// LMC_PacDrive/Application/TemplateFullProgrammingFramework/Visualization/Multicarrier/Vis_Positions_31_60
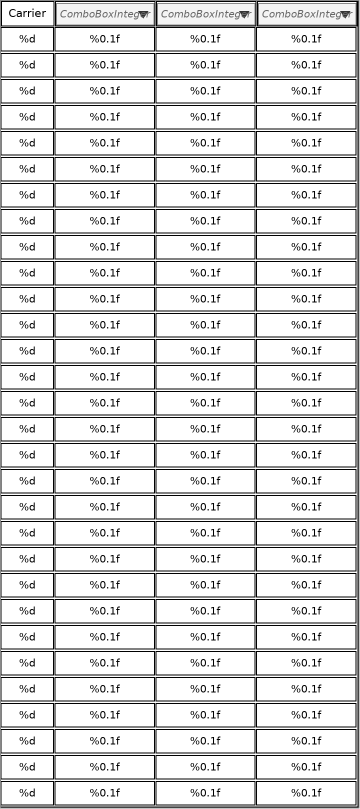
VISUALIZATION Vis_Positions_31_60  // 360x809
    Rectangle (0,0 358x807)
    Rectangle (55,1 100x25), "Position", invisible if: not SR_MultiCarriermodule.xInitSuccessful
    Rectangle (156,1 100x25), "Gap In Front", invisible if: not SR_MultiCarriermodule.xInitSuccessful
    Rectangle (257,1 100x25), "Gap Behind", invisible if: not SR_MultiCarriermodule.xInitSuccessful
    Rectangle (1,1 53x25), "Carrier", invisible if: not SR_MultiCarriermodule.xInitSuccessful
    Frame (0,27 358x26), invisible if: SR_MulticarrierModule.ifMulticarrier.ifFeedback.ifFeedbackConfiguration.udiNumberOfCarriers < 31 OR NOT SR_MultiCarriermodule.xInitSuccessful
        shows FR_CarDist(i_ifCarrierFeedback := SR_MultiCarrierModule.aifVisFeedback[31])
    Frame (0,53 358x26), invisible if: SR_MulticarrierModule.ifMulticarrier.ifFeedback.ifFeedbackConfiguration.udiNumberOfCarriers < 32 OR NOT SR_MultiCarriermodule.xInitSuccessful
        shows FR_CarDist(i_ifCarrierFeedback := SR_MultiCarrierModule.aifVisFeedback[32])
    Frame (0,79 358x26), invisible if: SR_MulticarrierModule.ifMulticarrier.ifFeedback.ifFeedbackConfiguration.udiNumberOfCarriers < 33 OR NOT SR_MultiCarriermodule.xInitSuccessful
        shows FR_CarDist(i_ifCarrierFeedback := SR_MultiCarrierModule.aifVisFeedback[33])
    Frame (0,105 358x26), invisible if: SR_MulticarrierModule.ifMulticarrier.ifFeedback.ifFeedbackConfiguration.udiNumberOfCarriers < 34 OR NOT SR_MultiCarriermodule.xInitSuccessful
        shows FR_CarDist(i_ifCarrierFeedback := SR_MultiCarrierModule.aifVisFeedback[34])
    Frame (0,131 358x26), invisible if: SR_MulticarrierModule.ifMulticarrier.ifFeedback.ifFeedbackConfiguration.udiNumberOfCarriers < 35 OR NOT SR_MultiCarriermodule.xInitSuccessful
        shows FR_CarDist(i_ifCarrierFeedback := SR_MultiCarrierModule.aifVisFeedback[35])
    Frame (0,157 358x26), invisible if: SR_MulticarrierModule.ifMulticarrier.ifFeedback.ifFeedbackConfiguration.udiNumberOfCarriers < 36 OR NOT SR_MultiCarriermodule.xInitSuccessful
        shows FR_CarDist(i_ifCarrierFeedback := SR_MultiCarrierModule.aifVisFeedback[36])
    Frame (0,183 358x26), invisible if: SR_MulticarrierModule.ifMulticarrier.ifFeedback.ifFeedbackConfiguration.udiNumberOfCarriers < 37 OR NOT SR_MultiCarriermodule.xInitSuccessful
        shows FR_CarDist(i_ifCarrierFeedback := SR_MultiCarrierModule.aifVisFeedback[37])
    Frame (0,209 358x26), invisible if: SR_MulticarrierModule.ifMulticarrier.ifFeedback.ifFeedbackConfiguration.udiNumberOfCarriers < 38 OR NOT SR_MultiCarriermodule.xInitSuccessful
        shows FR_CarDist(i_ifCarrierFeedback := SR_MultiCarrierModule.aifVisFeedback[38])
    Frame (0,235 358x26), invisible if: SR_MulticarrierModule.ifMulticarrier.ifFeedback.ifFeedbackConfiguration.udiNumberOfCarriers < 39 OR NOT SR_MultiCarriermodule.xInitSuccessful
        shows FR_CarDist(i_ifCarrierFeedback := SR_MultiCarrierModule.aifVisFeedback[39])
    Frame (0,261 358x26), invisible if: SR_MulticarrierModule.ifMulticarrier.ifFeedback.ifFeedbackConfiguration.udiNumberOfCarriers < 40 OR NOT SR_MultiCarriermodule.xInitSuccessful
        shows FR_CarDist(i_ifCarrierFeedback := SR_MultiCarrierModule.aifVisFeedback[40])
    ComboBoxInteger (258,3 98x22), tooltip "RefTrackPosition RefPosition Gap to Carrier in front Distance to Carrier in front Gap to Carrier behind Distance to Carrier behind", variable: SR_MulticarrierModule.etVisPosColumn3, text list: 'TextList_VisPositions'
    ComboBoxInteger (157,3 98x22), tooltip "RefTrackPosition RefPosition Gap to Carrier in front Distance to Carrier in front Gap to Carrier behind Distance to Carrier behind", variable: SR_MulticarrierModule.etVisPosColumn2, text list: 'TextList_VisPositions'
    ComboBoxInteger (56,3 98x22), tooltip "RefTrackPosition RefPosition Gap to Carrier in front Distance to Carrier in front Gap to Carrier behind Distance to Carrier behind", variable: SR_MulticarrierModule.etVisPosColumn1, text list: 'TextList_VisPositions'
    Frame (0,495 358x26), invisible if: SR_MulticarrierModule.ifMulticarrier.ifFeedback.ifFeedbackConfiguration.udiNumberOfCarriers < 50 OR NOT SR_MultiCarriermodule.xInitSuccessful
        shows FR_CarDist(i_ifCarrierFeedback := SR_MultiCarrierModule.aifVisFeedback[50])
    Frame (0,547 358x26), invisible if: SR_MulticarrierModule.ifMulticarrier.ifFeedback.ifFeedbackConfiguration.udiNumberOfCarriers < 51 OR NOT SR_MultiCarriermodule.xInitSuccessful
        shows FR_CarDist(i_ifCarrierFeedback := SR_MultiCarrierModule.aifVisFeedback[51])
    Frame (0,573 358x26), invisible if: SR_MulticarrierModule.ifMulticarrier.ifFeedback.ifFeedbackConfiguration.udiNumberOfCarriers < 52 OR NOT SR_MultiCarriermodule.xInitSuccessful
        shows FR_CarDist(i_ifCarrierFeedback := SR_MultiCarrierModule.aifVisFeedback[52])
    Frame (0,599 358x26), invisible if: SR_MulticarrierModule.ifMulticarrier.ifFeedback.ifFeedbackConfiguration.udiNumberOfCarriers < 53 OR NOT SR_MultiCarriermodule.xInitSuccessful
        shows FR_CarDist(i_ifCarrierFeedback := SR_MultiCarrierModule.aifVisFeedback[53])
    Frame (0,625 358x26), invisible if: SR_MulticarrierModule.ifMulticarrier.ifFeedback.ifFeedbackConfiguration.udiNumberOfCarriers < 54 OR NOT SR_MultiCarriermodule.xInitSuccessful
        shows FR_CarDist(i_ifCarrierFeedback := SR_MultiCarrierModule.aifVisFeedback[54])
    Frame (0,651 358x26), invisible if: SR_MulticarrierModule.ifMulticarrier.ifFeedback.ifFeedbackConfiguration.udiNumberOfCarriers < 55 OR NOT SR_MultiCarriermodule.xInitSuccessful
        shows FR_CarDist(i_ifCarrierFeedback := SR_MultiCarrierModule.aifVisFeedback[55])
    Frame (0,677 358x26), invisible if: SR_MulticarrierModule.ifMulticarrier.ifFeedback.ifFeedbackConfiguration.udiNumberOfCarriers < 56 OR NOT SR_MultiCarriermodule.xInitSuccessful
        shows FR_CarDist(i_ifCarrierFeedback := SR_MultiCarrierModule.aifVisFeedback[56])
    Frame (0,703 358x26), invisible if: SR_MulticarrierModule.ifMulticarrier.ifFeedback.ifFeedbackConfiguration.udiNumberOfCarriers < 57 OR NOT SR_MultiCarriermodule.xInitSuccessful
        shows FR_CarDist(i_ifCarrierFeedback := SR_MultiCarrierModule.aifVisFeedback[57])
    Frame (0,729 358x26), invisible if: SR_MulticarrierModule.ifMulticarrier.ifFeedback.ifFeedbackConfiguration.udiNumberOfCarriers < 58 OR NOT SR_MultiCarriermodule.xInitSuccessful
        shows FR_CarDist(i_ifCarrierFeedback := SR_MultiCarrierModule.aifVisFeedback[58])
    Frame (0,755 358x26), invisible if: SR_MulticarrierModule.ifMulticarrier.ifFeedback.ifFeedbackConfiguration.udiNumberOfCarriers < 59 OR NOT SR_MultiCarriermodule.xInitSuccessful
        shows FR_CarDist(i_ifCarrierFeedback := SR_MultiCarrierModule.aifVisFeedback[59])
    Frame (0,287 358x26), invisible if: SR_MulticarrierModule.ifMulticarrier.ifFeedback.ifFeedbackConfiguration.udiNumberOfCarriers < 41 OR NOT SR_MultiCarriermodule.xInitSuccessful
        shows FR_CarDist(i_ifCarrierFeedback := SR_MultiCarrierModule.aifVisFeedback[41])
    Frame (0,313 358x26), invisible if: SR_MulticarrierModule.ifMulticarrier.ifFeedback.ifFeedbackConfiguration.udiNumberOfCarriers < 42 OR NOT SR_MultiCarriermodule.xInitSuccessful
        shows FR_CarDist(i_ifCarrierFeedback := SR_MultiCarrierModule.aifVisFeedback[42])
    Frame (0,339 358x26), invisible if: SR_MulticarrierModule.ifMulticarrier.ifFeedback.ifFeedbackConfiguration.udiNumberOfCarriers < 43 OR NOT SR_MultiCarriermodule.xInitSuccessful
        shows FR_CarDist(i_ifCarrierFeedback := SR_MultiCarrierModule.aifVisFeedback[43])
    Frame (0,365 358x26), invisible if: SR_MulticarrierModule.ifMulticarrier.ifFeedback.ifFeedbackConfiguration.udiNumberOfCarriers < 44 OR NOT SR_MultiCarriermodule.xInitSuccessful
        shows FR_CarDist(i_ifCarrierFeedback := SR_MultiCarrierModule.aifVisFeedback[44])
    Frame (0,391 358x26), invisible if: SR_MulticarrierModule.ifMulticarrier.ifFeedback.ifFeedbackConfiguration.udiNumberOfCarriers < 45 OR NOT SR_MultiCarriermodule.xInitSuccessful
        shows FR_CarDist(i_ifCarrierFeedback := SR_MultiCarrierModule.aifVisFeedback[45])
    Frame (0,417 358x26), invisible if: SR_MulticarrierModule.ifMulticarrier.ifFeedback.ifFeedbackConfiguration.udiNumberOfCarriers < 46 OR NOT SR_MultiCarriermodule.xInitSuccessful
        shows FR_CarDist(i_ifCarrierFeedback := SR_MultiCarrierModule.aifVisFeedback[46])
    Frame (0,443 358x26), invisible if: SR_MulticarrierModule.ifMulticarrier.ifFeedback.ifFeedbackConfiguration.udiNumberOfCarriers < 47 OR NOT SR_MultiCarriermodule.xInitSuccessful
        shows FR_CarDist(i_ifCarrierFeedback := SR_MultiCarrierModule.aifVisFeedback[47])
    Frame (0,469 358x26), invisible if: SR_MulticarrierModule.ifMulticarrier.ifFeedback.ifFeedbackConfiguration.udiNumberOfCarriers < 48 OR NOT SR_MultiCarriermodule.xInitSuccessful
        shows FR_CarDist(i_ifCarrierFeedback := SR_MultiCarrierModule.aifVisFeedback[48])
    Frame (0,495 358x26), invisible if: SR_MulticarrierModule.ifMulticarrier.ifFeedback.ifFeedbackConfiguration.udiNumberOfCarriers < 49 OR NOT SR_MultiCarriermodule.xInitSuccessful
        shows FR_CarDist(i_ifCarrierFeedback := SR_MultiCarrierModule.aifVisFeedback[49])
    Frame (0,521 358x26), invisible if: SR_MulticarrierModule.ifMulticarrier.ifFeedback.ifFeedbackConfiguration.udiNumberOfCarriers < 50 OR NOT SR_MultiCarriermodule.xInitSuccessful
        shows FR_CarDist(i_ifCarrierFeedback := SR_MultiCarrierModule.aifVisFeedback[50])
    Frame (0,781 358x26), invisible if: SR_MulticarrierModule.ifMulticarrier.ifFeedback.ifFeedbackConfiguration.udiNumberOfCarriers < 60 OR NOT SR_MultiCarriermodule.xInitSuccessful
        shows FR_CarDist(i_ifCarrierFeedback := SR_MultiCarrierModule.aifVisFeedback[60])
END_VISUALIZATION

// LMC_PacDrive/Application/TemplateFullProgrammingFramework/Visualization/Multicarrier/Vis_Positions_61_90
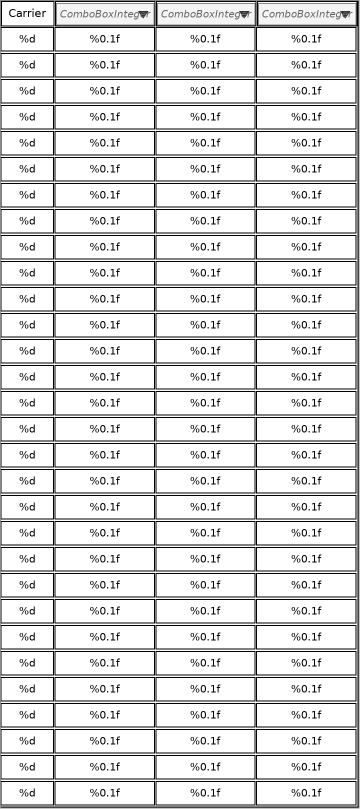
VISUALIZATION Vis_Positions_61_90  // 360x809
    Rectangle (0,0 358x807)
    Rectangle (55,1 100x25), "Position", invisible if: not SR_MultiCarriermodule.xInitSuccessful
    Rectangle (156,1 100x25), "Gap In Front", invisible if: not SR_MultiCarriermodule.xInitSuccessful
    Rectangle (257,1 100x25), "Gap Behind", invisible if: not SR_MultiCarriermodule.xInitSuccessful
    Rectangle (1,1 53x25), "Carrier", invisible if: not SR_MultiCarriermodule.xInitSuccessful
    Rectangle (55,1 100x25), "Position", invisible if: not SR_MultiCarriermodule.xInitSuccessful
    Rectangle (156,1 100x25), "Gap In Front", invisible if: not SR_MultiCarriermodule.xInitSuccessful
    Rectangle (257,1 100x25), "Gap Behind", invisible if: not SR_MultiCarriermodule.xInitSuccessful
    ComboBoxInteger (258,3 98x22), tooltip "RefTrackPosition RefPosition Gap to Carrier in front Distance to Carrier in front Gap to Carrier behind Distance to Carrier behind", variable: SR_MulticarrierModule.etVisPosColumn3, text list: 'TextList_VisPositions'
    ComboBoxInteger (157,3 98x22), tooltip "RefTrackPosition RefPosition Gap to Carrier in front Distance to Carrier in front Gap to Carrier behind Distance to Carrier behind", variable: SR_MulticarrierModule.etVisPosColumn2, text list: 'TextList_VisPositions'
    ComboBoxInteger (56,3 98x22), tooltip "RefTrackPosition RefPosition Gap to Carrier in front Distance to Carrier in front Gap to Carrier behind Distance to Carrier behind", variable: SR_MulticarrierModule.etVisPosColumn1, text list: 'TextList_VisPositions'
    Frame (0,27 358x26), invisible if: SR_MulticarrierModule.ifMulticarrier.ifFeedback.ifFeedbackConfiguration.udiNumberOfCarriers < 61 OR NOT SR_MultiCarriermodule.xInitSuccessful
        shows FR_CarDist(i_ifCarrierFeedback := SR_MultiCarrierModule.aifVisFeedback[61])
    Frame (0,261 358x26), invisible if: SR_MulticarrierModule.ifMulticarrier.ifFeedback.ifFeedbackConfiguration.udiNumberOfCarriers < 70 OR NOT SR_MultiCarriermodule.xInitSuccessful
        shows FR_CarDist(i_ifCarrierFeedback := SR_MultiCarrierModule.aifVisFeedback[70])
    Frame (0,53 358x26), invisible if: SR_MulticarrierModule.ifMulticarrier.ifFeedback.ifFeedbackConfiguration.udiNumberOfCarriers < 62 OR NOT SR_MultiCarriermodule.xInitSuccessful
        shows FR_CarDist(i_ifCarrierFeedback := SR_MultiCarrierModule.aifVisFeedback[62])
    Frame (0,105 358x26), invisible if: SR_MulticarrierModule.ifMulticarrier.ifFeedback.ifFeedbackConfiguration.udiNumberOfCarriers < 64 OR NOT SR_MultiCarriermodule.xInitSuccessful
        shows FR_CarDist(i_ifCarrierFeedback := SR_MultiCarrierModule.aifVisFeedback[64])
    Frame (0,131 358x26), invisible if: SR_MulticarrierModule.ifMulticarrier.ifFeedback.ifFeedbackConfiguration.udiNumberOfCarriers < 65 OR NOT SR_MultiCarriermodule.xInitSuccessful
        shows FR_CarDist(i_ifCarrierFeedback := SR_MultiCarrierModule.aifVisFeedback[65])
    Frame (0,157 358x26), invisible if: SR_MulticarrierModule.ifMulticarrier.ifFeedback.ifFeedbackConfiguration.udiNumberOfCarriers < 66 OR NOT SR_MultiCarriermodule.xInitSuccessful
        shows FR_CarDist(i_ifCarrierFeedback := SR_MultiCarrierModule.aifVisFeedback[66])
    Frame (0,209 358x26), invisible if: SR_MulticarrierModule.ifMulticarrier.ifFeedback.ifFeedbackConfiguration.udiNumberOfCarriers < 68 OR NOT SR_MultiCarriermodule.xInitSuccessful
        shows FR_CarDist(i_ifCarrierFeedback := SR_MultiCarrierModule.aifVisFeedback[68])
    Frame (0,235 358x26), invisible if: SR_MulticarrierModule.ifMulticarrier.ifFeedback.ifFeedbackConfiguration.udiNumberOfCarriers < 69 OR NOT SR_MultiCarriermodule.xInitSuccessful
        shows FR_CarDist(i_ifCarrierFeedback := SR_MultiCarrierModule.aifVisFeedback[69])
    Frame (0,287 358x26), invisible if: SR_MulticarrierModule.ifMulticarrier.ifFeedback.ifFeedbackConfiguration.udiNumberOfCarriers < 71 OR NOT SR_MultiCarriermodule.xInitSuccessful
        shows FR_CarDist(i_ifCarrierFeedback := SR_MultiCarrierModule.aifVisFeedback[71])
    Frame (0,313 358x26), invisible if: SR_MulticarrierModule.ifMulticarrier.ifFeedback.ifFeedbackConfiguration.udiNumberOfCarriers < 72 OR NOT SR_MultiCarriermodule.xInitSuccessful
        shows FR_CarDist(i_ifCarrierFeedback := SR_MultiCarrierModule.aifVisFeedback[72])
    Frame (0,339 358x26), invisible if: SR_MulticarrierModule.ifMulticarrier.ifFeedback.ifFeedbackConfiguration.udiNumberOfCarriers < 73 OR NOT SR_MultiCarriermodule.xInitSuccessful
        shows FR_CarDist(i_ifCarrierFeedback := SR_MultiCarrierModule.aifVisFeedback[73])
    Frame (0,365 358x26), invisible if: SR_MulticarrierModule.ifMulticarrier.ifFeedback.ifFeedbackConfiguration.udiNumberOfCarriers < 74 OR NOT SR_MultiCarriermodule.xInitSuccessful
        shows FR_CarDist(i_ifCarrierFeedback := SR_MultiCarrierModule.aifVisFeedback[74])
    Frame (0,391 358x26), invisible if: SR_MulticarrierModule.ifMulticarrier.ifFeedback.ifFeedbackConfiguration.udiNumberOfCarriers < 75 OR NOT SR_MultiCarriermodule.xInitSuccessful
        shows FR_CarDist(i_ifCarrierFeedback := SR_MultiCarrierModule.aifVisFeedback[75])
    Frame (0,417 358x26), invisible if: SR_MulticarrierModule.ifMulticarrier.ifFeedback.ifFeedbackConfiguration.udiNumberOfCarriers < 76 OR NOT SR_MultiCarriermodule.xInitSuccessful
        shows FR_CarDist(i_ifCarrierFeedback := SR_MultiCarrierModule.aifVisFeedback[76])
    Frame (0,443 358x26), invisible if: SR_MulticarrierModule.ifMulticarrier.ifFeedback.ifFeedbackConfiguration.udiNumberOfCarriers < 77 OR NOT SR_MultiCarriermodule.xInitSuccessful
        shows FR_CarDist(i_ifCarrierFeedback := SR_MultiCarrierModule.aifVisFeedback[77])
    Frame (0,469 358x26), invisible if: SR_MulticarrierModule.ifMulticarrier.ifFeedback.ifFeedbackConfiguration.udiNumberOfCarriers < 78 OR NOT SR_MultiCarriermodule.xInitSuccessful
        shows FR_CarDist(i_ifCarrierFeedback := SR_MultiCarrierModule.aifVisFeedback[78])
    Frame (0,495 358x26), invisible if: SR_MulticarrierModule.ifMulticarrier.ifFeedback.ifFeedbackConfiguration.udiNumberOfCarriers < 79 OR NOT SR_MultiCarriermodule.xInitSuccessful
        shows FR_CarDist(i_ifCarrierFeedback := SR_MultiCarrierModule.aifVisFeedback[79])
    Frame (0,521 358x26), invisible if: SR_MulticarrierModule.ifMulticarrier.ifFeedback.ifFeedbackConfiguration.udiNumberOfCarriers < 80 OR NOT SR_MultiCarriermodule.xInitSuccessful
        shows FR_CarDist(i_ifCarrierFeedback := SR_MultiCarrierModule.aifVisFeedback[80])
    Frame (0,79 358x26), invisible if: SR_MulticarrierModule.ifMulticarrier.ifFeedback.ifFeedbackConfiguration.udiNumberOfCarriers < 63 OR NOT SR_MultiCarriermodule.xInitSuccessful
        shows FR_CarDist(i_ifCarrierFeedback := SR_MultiCarrierModule.aifVisFeedback[63])
    Frame (0,183 358x26), invisible if: SR_MulticarrierModule.ifMulticarrier.ifFeedback.ifFeedbackConfiguration.udiNumberOfCarriers < 67 OR NOT SR_MultiCarriermodule.xInitSuccessful
        shows FR_CarDist(i_ifCarrierFeedback := SR_MultiCarrierModule.aifVisFeedback[67])
    Frame (0,547 358x26), invisible if: SR_MulticarrierModule.ifMulticarrier.ifFeedback.ifFeedbackConfiguration.udiNumberOfCarriers < 81 OR NOT SR_MultiCarriermodule.xInitSuccessful
        shows FR_CarDist(i_ifCarrierFeedback := SR_MultiCarrierModule.aifVisFeedback[81])
    Frame (0,573 358x26), invisible if: SR_MulticarrierModule.ifMulticarrier.ifFeedback.ifFeedbackConfiguration.udiNumberOfCarriers < 82 OR NOT SR_MultiCarriermodule.xInitSuccessful
        shows FR_CarDist(i_ifCarrierFeedback := SR_MultiCarrierModule.aifVisFeedback[82])
    Frame (0,599 358x26), invisible if: SR_MulticarrierModule.ifMulticarrier.ifFeedback.ifFeedbackConfiguration.udiNumberOfCarriers < 83 OR NOT SR_MultiCarriermodule.xInitSuccessful
        shows FR_CarDist(i_ifCarrierFeedback := SR_MultiCarrierModule.aifVisFeedback[83])
    Frame (0,625 358x26), invisible if: SR_MulticarrierModule.ifMulticarrier.ifFeedback.ifFeedbackConfiguration.udiNumberOfCarriers < 84 OR NOT SR_MultiCarriermodule.xInitSuccessful
        shows FR_CarDist(i_ifCarrierFeedback := SR_MultiCarrierModule.aifVisFeedback[84])
    Frame (0,651 358x26), invisible if: SR_MulticarrierModule.ifMulticarrier.ifFeedback.ifFeedbackConfiguration.udiNumberOfCarriers < 85 OR NOT SR_MultiCarriermodule.xInitSuccessful
        shows FR_CarDist(i_ifCarrierFeedback := SR_MultiCarrierModule.aifVisFeedback[85])
    Frame (0,677 358x26), invisible if: SR_MulticarrierModule.ifMulticarrier.ifFeedback.ifFeedbackConfiguration.udiNumberOfCarriers < 86 OR NOT SR_MultiCarriermodule.xInitSuccessful
        shows FR_CarDist(i_ifCarrierFeedback := SR_MultiCarrierModule.aifVisFeedback[86])
    Frame (0,703 358x26), invisible if: SR_MulticarrierModule.ifMulticarrier.ifFeedback.ifFeedbackConfiguration.udiNumberOfCarriers < 87 OR NOT SR_MultiCarriermodule.xInitSuccessful
        shows FR_CarDist(i_ifCarrierFeedback := SR_MultiCarrierModule.aifVisFeedback[87])
    Frame (0,729 358x26), invisible if: SR_MulticarrierModule.ifMulticarrier.ifFeedback.ifFeedbackConfiguration.udiNumberOfCarriers < 88 OR NOT SR_MultiCarriermodule.xInitSuccessful
        shows FR_CarDist(i_ifCarrierFeedback := SR_MultiCarrierModule.aifVisFeedback[88])
    Frame (0,755 358x26), invisible if: SR_MulticarrierModule.ifMulticarrier.ifFeedback.ifFeedbackConfiguration.udiNumberOfCarriers < 89 OR NOT SR_MultiCarriermodule.xInitSuccessful
        shows FR_CarDist(i_ifCarrierFeedback := SR_MultiCarrierModule.aifVisFeedback[89])
    Frame (0,781 358x26), invisible if: SR_MulticarrierModule.ifMulticarrier.ifFeedback.ifFeedbackConfiguration.udiNumberOfCarriers < 90 OR NOT SR_MultiCarriermodule.xInitSuccessful
        shows FR_CarDist(i_ifCarrierFeedback := SR_MultiCarrierModule.aifVisFeedback[90])
END_VISUALIZATION

// LMC_PacDrive/Application/TemplateFullProgrammingFramework/Visualization/Multicarrier/Vis_Positions_91_120
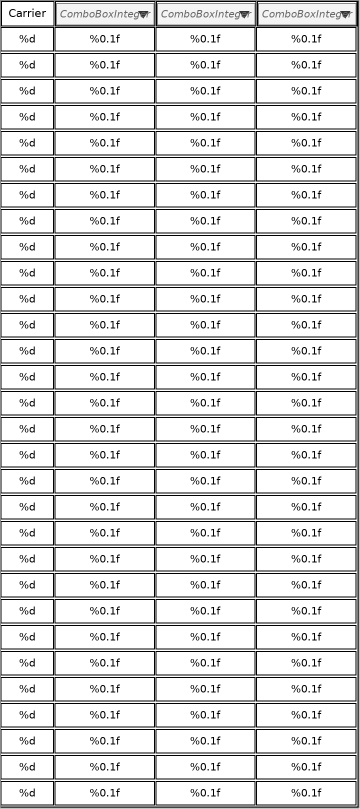
VISUALIZATION Vis_Positions_91_120  // 360x809
    Rectangle (0,0 358x807)
    Rectangle (55,1 100x25), "Position"
    Rectangle (257,1 100x25), "Gap Behind"
    Rectangle (1,1 53x25), "Carrier"
    Rectangle (156,1 100x25), "Gap In Front"
    Rectangle (55,1 100x25), "Position", invisible if: not SR_MultiCarriermodule.xInitSuccessful
    Rectangle (156,1 100x25), "Gap In Front", invisible if: not SR_MultiCarriermodule.xInitSuccessful
    Rectangle (257,1 100x25), "Gap Behind", invisible if: not SR_MultiCarriermodule.xInitSuccessful
    ComboBoxInteger (258,3 98x22), tooltip "RefTrackPosition RefPosition Gap to Carrier in front Distance to Carrier in front Gap to Carrier behind Distance to Carrier behind", variable: SR_MulticarrierModule.etVisPosColumn3, text list: 'TextList_VisPositions'
    ComboBoxInteger (157,3 98x22), tooltip "RefTrackPosition RefPosition Gap to Carrier in front Distance to Carrier in front Gap to Carrier behind Distance to Carrier behind", variable: SR_MulticarrierModule.etVisPosColumn2, text list: 'TextList_VisPositions'
    ComboBoxInteger (56,3 98x22), tooltip "RefTrackPosition RefPosition Gap to Carrier in front Distance to Carrier in front Gap to Carrier behind Distance to Carrier behind", variable: SR_MulticarrierModule.etVisPosColumn1, text list: 'TextList_VisPositions'
    Frame (0,261 358x26), invisible if: SR_MulticarrierModule.ifMulticarrier.ifFeedback.ifFeedbackConfiguration.udiNumberOfCarriers < 100 OR NOT SR_MultiCarriermodule.xInitSuccessful
        shows FR_CarDist(i_ifCarrierFeedback := SR_MultiCarrierModule.aifVisFeedback[100])
    Frame (0,287 358x26), invisible if: SR_MulticarrierModule.ifMulticarrier.ifFeedback.ifFeedbackConfiguration.udiNumberOfCarriers < 101 OR NOT SR_MultiCarriermodule.xInitSuccessful
        shows FR_CarDist(i_ifCarrierFeedback := SR_MultiCarrierModule.aifVisFeedback[101])
    Frame (0,313 358x26), invisible if: SR_MulticarrierModule.ifMulticarrier.ifFeedback.ifFeedbackConfiguration.udiNumberOfCarriers < 102 OR NOT SR_MultiCarriermodule.xInitSuccessful
        shows FR_CarDist(i_ifCarrierFeedback := SR_MultiCarrierModule.aifVisFeedback[102])
    Frame (0,339 358x26), invisible if: SR_MulticarrierModule.ifMulticarrier.ifFeedback.ifFeedbackConfiguration.udiNumberOfCarriers < 103 OR NOT SR_MultiCarriermodule.xInitSuccessful
        shows FR_CarDist(i_ifCarrierFeedback := SR_MultiCarrierModule.aifVisFeedback[103])
    Frame (0,365 358x26), invisible if: SR_MulticarrierModule.ifMulticarrier.ifFeedback.ifFeedbackConfiguration.udiNumberOfCarriers < 104 OR NOT SR_MultiCarriermodule.xInitSuccessful
        shows FR_CarDist(i_ifCarrierFeedback := SR_MultiCarrierModule.aifVisFeedback[104])
    Frame (0,391 358x26), invisible if: SR_MulticarrierModule.ifMulticarrier.ifFeedback.ifFeedbackConfiguration.udiNumberOfCarriers < 105 OR NOT SR_MultiCarriermodule.xInitSuccessful
        shows FR_CarDist(i_ifCarrierFeedback := SR_MultiCarrierModule.aifVisFeedback[105])
    Frame (0,417 358x26), invisible if: SR_MulticarrierModule.ifMulticarrier.ifFeedback.ifFeedbackConfiguration.udiNumberOfCarriers < 106 OR NOT SR_MultiCarriermodule.xInitSuccessful
        shows FR_CarDist(i_ifCarrierFeedback := SR_MultiCarrierModule.aifVisFeedback[106])
    Frame (0,443 358x26), invisible if: SR_MulticarrierModule.ifMulticarrier.ifFeedback.ifFeedbackConfiguration.udiNumberOfCarriers < 107 OR NOT SR_MultiCarriermodule.xInitSuccessful
        shows FR_CarDist(i_ifCarrierFeedback := SR_MultiCarrierModule.aifVisFeedback[107])
    Frame (0,469 358x26), invisible if: SR_MulticarrierModule.ifMulticarrier.ifFeedback.ifFeedbackConfiguration.udiNumberOfCarriers < 108 OR NOT SR_MultiCarriermodule.xInitSuccessful
        shows FR_CarDist(i_ifCarrierFeedback := SR_MultiCarrierModule.aifVisFeedback[108])
    Frame (0,495 358x26), invisible if: SR_MulticarrierModule.ifMulticarrier.ifFeedback.ifFeedbackConfiguration.udiNumberOfCarriers < 109 OR NOT SR_MultiCarriermodule.xInitSuccessful
        shows FR_CarDist(i_ifCarrierFeedback := SR_MultiCarrierModule.aifVisFeedback[109])
    Frame (0,521 358x26), invisible if: SR_MulticarrierModule.ifMulticarrier.ifFeedback.ifFeedbackConfiguration.udiNumberOfCarriers < 110 OR NOT SR_MultiCarriermodule.xInitSuccessful
        shows FR_CarDist(i_ifCarrierFeedback := SR_MultiCarrierModule.aifVisFeedback[110])
    Frame (0,547 358x26), invisible if: SR_MulticarrierModule.ifMulticarrier.ifFeedback.ifFeedbackConfiguration.udiNumberOfCarriers < 111 OR NOT SR_MultiCarriermodule.xInitSuccessful
        shows FR_CarDist(i_ifCarrierFeedback := SR_MultiCarrierModule.aifVisFeedback[111])
    Frame (0,573 358x26), invisible if: SR_MulticarrierModule.ifMulticarrier.ifFeedback.ifFeedbackConfiguration.udiNumberOfCarriers < 112 OR NOT SR_MultiCarriermodule.xInitSuccessful
        shows FR_CarDist(i_ifCarrierFeedback := SR_MultiCarrierModule.aifVisFeedback[112])
    Frame (0,599 358x26), invisible if: SR_MulticarrierModule.ifMulticarrier.ifFeedback.ifFeedbackConfiguration.udiNumberOfCarriers < 113 OR NOT SR_MultiCarriermodule.xInitSuccessful
        shows FR_CarDist(i_ifCarrierFeedback := SR_MultiCarrierModule.aifVisFeedback[113])
    Frame (0,625 358x26), invisible if: SR_MulticarrierModule.ifMulticarrier.ifFeedback.ifFeedbackConfiguration.udiNumberOfCarriers < 114 OR NOT SR_MultiCarriermodule.xInitSuccessful
        shows FR_CarDist(i_ifCarrierFeedback := SR_MultiCarrierModule.aifVisFeedback[114])
    Frame (0,651 358x26), invisible if: SR_MulticarrierModule.ifMulticarrier.ifFeedback.ifFeedbackConfiguration.udiNumberOfCarriers < 115 OR NOT SR_MultiCarriermodule.xInitSuccessful
        shows FR_CarDist(i_ifCarrierFeedback := SR_MultiCarrierModule.aifVisFeedback[115])
    Frame (0,677 358x26), invisible if: SR_MulticarrierModule.ifMulticarrier.ifFeedback.ifFeedbackConfiguration.udiNumberOfCarriers < 116 OR NOT SR_MultiCarriermodule.xInitSuccessful
        shows FR_CarDist(i_ifCarrierFeedback := SR_MultiCarrierModule.aifVisFeedback[116])
    Frame (0,703 358x26), invisible if: SR_MulticarrierModule.ifMulticarrier.ifFeedback.ifFeedbackConfiguration.udiNumberOfCarriers < 117 OR NOT SR_MultiCarriermodule.xInitSuccessful
        shows FR_CarDist(i_ifCarrierFeedback := SR_MultiCarrierModule.aifVisFeedback[117])
    Frame (0,729 358x26), invisible if: SR_MulticarrierModule.ifMulticarrier.ifFeedback.ifFeedbackConfiguration.udiNumberOfCarriers < 118 OR NOT SR_MultiCarriermodule.xInitSuccessful
        shows FR_CarDist(i_ifCarrierFeedback := SR_MultiCarrierModule.aifVisFeedback[118])
    Frame (0,755 358x26), invisible if: SR_MulticarrierModule.ifMulticarrier.ifFeedback.ifFeedbackConfiguration.udiNumberOfCarriers < 119 OR NOT SR_MultiCarriermodule.xInitSuccessful
        shows FR_CarDist(i_ifCarrierFeedback := SR_MultiCarrierModule.aifVisFeedback[119])
    Frame (0,781 358x26), invisible if: SR_MulticarrierModule.ifMulticarrier.ifFeedback.ifFeedbackConfiguration.udiNumberOfCarriers < 120 OR NOT SR_MultiCarriermodule.xInitSuccessful
        shows FR_CarDist(i_ifCarrierFeedback := SR_MultiCarrierModule.aifVisFeedback[120])
    Frame (0,27 358x26), invisible if: SR_MulticarrierModule.ifMulticarrier.ifFeedback.ifFeedbackConfiguration.udiNumberOfCarriers < 91 OR NOT SR_MultiCarriermodule.xInitSuccessful
        shows FR_CarDist(i_ifCarrierFeedback := SR_MultiCarrierModule.aifVisFeedback[91])
    Frame (0,53 358x26), invisible if: SR_MulticarrierModule.ifMulticarrier.ifFeedback.ifFeedbackConfiguration.udiNumberOfCarriers < 92 OR NOT SR_MultiCarriermodule.xInitSuccessful
        shows FR_CarDist(i_ifCarrierFeedback := SR_MultiCarrierModule.aifVisFeedback[92])
    Frame (0,79 358x26), invisible if: SR_MulticarrierModule.ifMulticarrier.ifFeedback.ifFeedbackConfiguration.udiNumberOfCarriers < 93 OR NOT SR_MultiCarriermodule.xInitSuccessful
        shows FR_CarDist(i_ifCarrierFeedback := SR_MultiCarrierModule.aifVisFeedback[93])
    Frame (0,105 358x26), invisible if: SR_MulticarrierModule.ifMulticarrier.ifFeedback.ifFeedbackConfiguration.udiNumberOfCarriers < 94 OR NOT SR_MultiCarriermodule.xInitSuccessful
        shows FR_CarDist(i_ifCarrierFeedback := SR_MultiCarrierModule.aifVisFeedback[94])
    Frame (0,131 358x26), invisible if: SR_MulticarrierModule.ifMulticarrier.ifFeedback.ifFeedbackConfiguration.udiNumberOfCarriers < 95 OR NOT SR_MultiCarriermodule.xInitSuccessful
        shows FR_CarDist(i_ifCarrierFeedback := SR_MultiCarrierModule.aifVisFeedback[95])
    Frame (0,157 358x26), invisible if: SR_MulticarrierModule.ifMulticarrier.ifFeedback.ifFeedbackConfiguration.udiNumberOfCarriers < 96 OR NOT SR_MultiCarriermodule.xInitSuccessful
        shows FR_CarDist(i_ifCarrierFeedback := SR_MultiCarrierModule.aifVisFeedback[96])
    Frame (0,183 358x26), invisible if: SR_MulticarrierModule.ifMulticarrier.ifFeedback.ifFeedbackConfiguration.udiNumberOfCarriers < 97 OR NOT SR_MultiCarriermodule.xInitSuccessful
        shows FR_CarDist(i_ifCarrierFeedback := SR_MultiCarrierModule.aifVisFeedback[97])
    Frame (0,209 358x26), invisible if: SR_MulticarrierModule.ifMulticarrier.ifFeedback.ifFeedbackConfiguration.udiNumberOfCarriers < 98 OR NOT SR_MultiCarriermodule.xInitSuccessful
        shows FR_CarDist(i_ifCarrierFeedback := SR_MultiCarrierModule.aifVisFeedback[98])
    Frame (0,235 358x26), invisible if: SR_MulticarrierModule.ifMulticarrier.ifFeedback.ifFeedbackConfiguration.udiNumberOfCarriers < 99 OR NOT SR_MultiCarriermodule.xInitSuccessful
        shows FR_CarDist(i_ifCarrierFeedback := SR_MultiCarrierModule.aifVisFeedback[99])
END_VISUALIZATION

// LMC_PacDrive/Application/TemplateFullProgrammingFramework/Visualization/Multicarrier/Vis_Trace
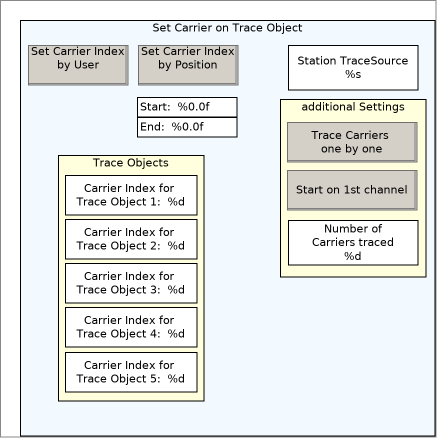
VISUALIZATION Vis_Trace  // 437x438
    Rectangle (20,20 415x416), "Set Carrier on Trace Object"
        OnMouseClick: write the text variable via Default
    Rectangle (280,99 146x178), "additional Settings", invisible if: SR_MultiCarriermodule.etTraceSource = ET_TraceSource.MultiCarriermodule or SR_MultiCarriermodule.etTraceSource = ET_TraceSource.StartPosAndEndPos
    Rectangle (288,220 130x45), "Number of Carriers traced %d", text variable: SR_MulticarrierModule.udiNumberOfCarrierInTrace, invisible if: SR_MultiCarriermodule.etTraceSource = ET_TraceSource.MultiCarriermodule or SR_MultiCarriermodule.etTraceSource = ET_TraceSource.StartPosAndEndPos, input disabled if: SR_MulticarrierModule.xOneByOne
        OnMouseClick: write the text variable via Default
    Rectangle (288,45 130x45), "Station TraceSource %s", text variable: SR_MulticarrierModule.etTraceSource, invisible if: SR_MultiCarriermodule.etTraceSource = ET_TraceSource.MultiCarriermodule or SR_MultiCarriermodule.etTraceSource = ET_TraceSource.StartPosAndEndPos, input disabled if: SR_MulticarrierModule.xOneByOne
    Button (28,45 100x40), "Set Carrier Index by User", colour toggle: SR_MultiCarriermodule.etTraceSource = ET_TraceSource.MultiCarriermodule
        OnMouseDown: execute { SR_MultiCarriermodule.etTraceSource := ET_TraceSource.MultiCarriermodule; }
    Button (287,122 130x40), "Trace Carriers one by one", colour toggle: SR_MulticarrierModule.xOneByOne, invisible if: SR_MultiCarriermodule.etTraceSource = ET_TraceSource.MultiCarriermodule or SR_MultiCarriermodule.etTraceSource = ET_TraceSource.StartPosAndEndPos
        toggle SR_MulticarrierModule.xOneByOne
    Button (287,170 130x40), "Start on 1st channel", invisible if: SR_MultiCarriermodule.etTraceSource = ET_TraceSource.MultiCarriermodule or SR_MultiCarriermodule.etTraceSource = ET_TraceSource.StartPosAndEndPos, input disabled if: SR_MulticarrierModule.xReStartOneByOneCount
        toggle SR_MulticarrierModule.xReStartOneByOneCount
    Rectangle (58,155 146x246), "Trace Objects", invisible if: not (SR_MultiCarriermodule.etTraceSource = ET_TraceSource.MulticarrierModule Or SR_MultiCarriermodule.etTraceSource = ET_TraceSource.StartPosAndEndPos )
        p2738717112: SR_MulticarrierModule.iTopTraceEntryVis
    Rectangle (65,175 132x40), "Carrier Index for Trace Object 1: %d", text variable: SR_MulticarrierModule.udiTraceObject1, invisible if: not (SR_MultiCarriermodule.etTraceSource = ET_TraceSource.MulticarrierModule Or SR_MultiCarriermodule.etTraceSource = ET_TraceSource.StartPosAndEndPos ), input disabled if: SR_MultiCarriermodule.etTraceSource = ET_TraceSource.StartPosAndEndPos
        p2738717112: SR_MulticarrierModule.iTopTraceEntryVis
        OnMouseClick: write the text variable via Default
    Rectangle (65,219 132x40), "Carrier Index for Trace Object 2: %d", text variable: SR_MulticarrierModule.udiTraceObject2, invisible if: not (SR_MultiCarriermodule.etTraceSource = ET_TraceSource.MulticarrierModule Or SR_MultiCarriermodule.etTraceSource = ET_TraceSource.StartPosAndEndPos ), input disabled if: SR_MultiCarriermodule.etTraceSource = ET_TraceSource.StartPosAndEndPos
        p2738717112: SR_MulticarrierModule.iTopTraceEntryVis
        OnMouseClick: write the text variable via Default
    Rectangle (65,263 132x40), "Carrier Index for Trace Object 3: %d", text variable: SR_MulticarrierModule.udiTraceObject3, invisible if: not (SR_MultiCarriermodule.etTraceSource = ET_TraceSource.MulticarrierModule Or SR_MultiCarriermodule.etTraceSource = ET_TraceSource.StartPosAndEndPos ), input disabled if: SR_MultiCarriermodule.etTraceSource = ET_TraceSource.StartPosAndEndPos
        p2738717112: SR_MulticarrierModule.iTopTraceEntryVis
        OnMouseClick: write the text variable via Default
    Rectangle (65,307 132x40), "Carrier Index for Trace Object 4: %d", text variable: SR_MulticarrierModule.udiTraceObject4, invisible if: not (SR_MultiCarriermodule.etTraceSource = ET_TraceSource.MulticarrierModule Or SR_MultiCarriermodule.etTraceSource = ET_TraceSource.StartPosAndEndPos ), input disabled if: SR_MultiCarriermodule.etTraceSource = ET_TraceSource.StartPosAndEndPos
        p2738717112: SR_MulticarrierModule.iTopTraceEntryVis
        OnMouseClick: write the text variable via Default
    Rectangle (65,352 132x40), "Carrier Index for Trace Object 5: %d", text variable: SR_MulticarrierModule.udiTraceObject5, invisible if: not (SR_MultiCarriermodule.etTraceSource = ET_TraceSource.MulticarrierModule Or SR_MultiCarriermodule.etTraceSource = ET_TraceSource.StartPosAndEndPos ), input disabled if: SR_MultiCarriermodule.etTraceSource = ET_TraceSource.StartPosAndEndPos
        p2738717112: SR_MulticarrierModule.iTopTraceEntryVis
        OnMouseClick: write the text variable via Default
    Button (138,45 100x40), "Set Carrier Index by Position", colour toggle: SR_MultiCarriermodule.etTraceSource = ET_TraceSource.StartPosAndEndPos
        OnMouseDown: execute { SR_MultiCarriermodule.etTraceSource := ET_TraceSource.StartPosAndEndPos; }
    Rectangle (137,97 100x20), "Start: %0.0f", text variable: SR_MulticarrierModule.lrTraceStartTrackPos, invisible if: not (SR_MultiCarriermodule.etTraceSource = ET_TraceSource.StartPosAndEndPos )
        OnMouseClick: write the text variable via Default, min 0, max SR_MulticarrierModule.fbMulticarrier.ifFeedback.ifFeedbackConfiguration.lrTrackLength
    Rectangle (137,117 100x20), "End: %0.0f", text variable: SR_MulticarrierModule.lrTraceEndTrackPos, invisible if: not (SR_MultiCarriermodule.etTraceSource = ET_TraceSource.StartPosAndEndPos )
        OnMouseClick: write the text variable via Default, min 0, max SR_MulticarrierModule.fbMulticarrier.ifFeedback.ifFeedbackConfiguration.lrTrackLength
END_VISUALIZATION

// LMC_PacDrive/Application/TemplateFullProgrammingFramework/Visualization/Multicarrier/Vis_TrackCalibration
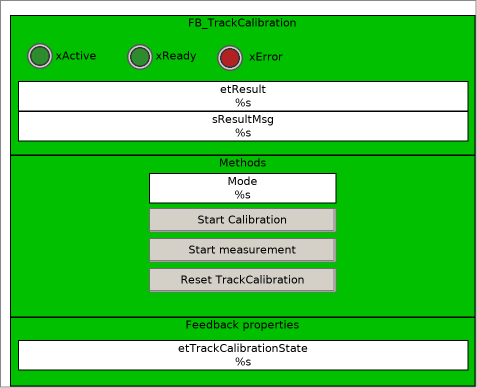
VISUALIZATION Vis_TrackCalibration  // 477x388
    Rectangle (10,15 465x140), "FB_TrackCalibration", invisible if: SR_PlayGround.xshowList, input disabled if: not SR_MainMachine.xActTrackCalibration
    Rectangle (10,155 465x162), "Methods"
    Rectangle (10,317 465x69), "Feedback properties"
    Rectangle (18,81 450x30), "etResult %s", text variable: SR_MulticarrierModule.etResultFbTrackCalibration, input disabled if: not SR_MainMachine.xActTrackCalibration
    Rectangle (18,111 450x30), "sResultMsg %s", text variable: SR_MulticarrierModule.sResultMsgFbTrackCalibration, input disabled if: not SR_MainMachine.xActTrackCalibration
    Rectangle (18,340 450x30), "etTrackCalibrationState %s", text variable: SR_MulticarrierModule.fbTrackCalibration.etState, input disabled if: not SR_MainMachine.xActTrackCalibration
    Button (149,208 187x24), "Start Calibration", input disabled if: not SR_MainMachine.xActTrackCalibration
        tap SR_MulticarrierModule.xStartCalibration
    Rectangle (54,41 44x30), "xActive", input disabled if: not SR_MainMachine.xActTrackCalibration
    Rectangle (154,41 44x30), "xReady", input disabled if: not SR_MainMachine.xActTrackCalibration
    Rectangle (244,42 44x30), "xError", input disabled if: not SR_MainMachine.xActTrackCalibration
    Line (10,155) (475,155)
    Lamp1 (25,41 30x30), variable: SR_MultiCarrierModule.xActiveFbTrackCalibration, style: Lamp-Lamp1-Green
    Lamp1 (125,42 30x30), variable: SR_MultiCarrierModule.xReadyFbTrackCalibration, style: Lamp-Lamp1-Green
    Lamp1 (215,43 30x30), variable: SR_MultiCarrierModule.xErrorFbTrackCalibration, style: Lamp-Lamp1-Red
    Button (149,268 187x24), "Reset TrackCalibration", input disabled if: not SR_MainMachine.xActTrackCalibration
        tap SR_MulticarrierModule.xResetTrackCalibration
    Button (149,238 187x24), "Start measurement", input disabled if: not SR_MainMachine.xActTrackCalibration
        tap SR_MulticarrierModule.xStartMeasurement
    Rectangle (149,173 187x30), "Mode %s", text variable: SR_MulticarrierModule.etModeTrackCalibration, input disabled if: not SR_MainMachine.xActTrackCalibration
        OnMouseClick: write the text variable via Default, min 0, max 2
END_VISUALIZATION

// LMC_PacDrive/Application/TemplateFullProgrammingFramework/Visualization/Windows/VIS_AxisModule
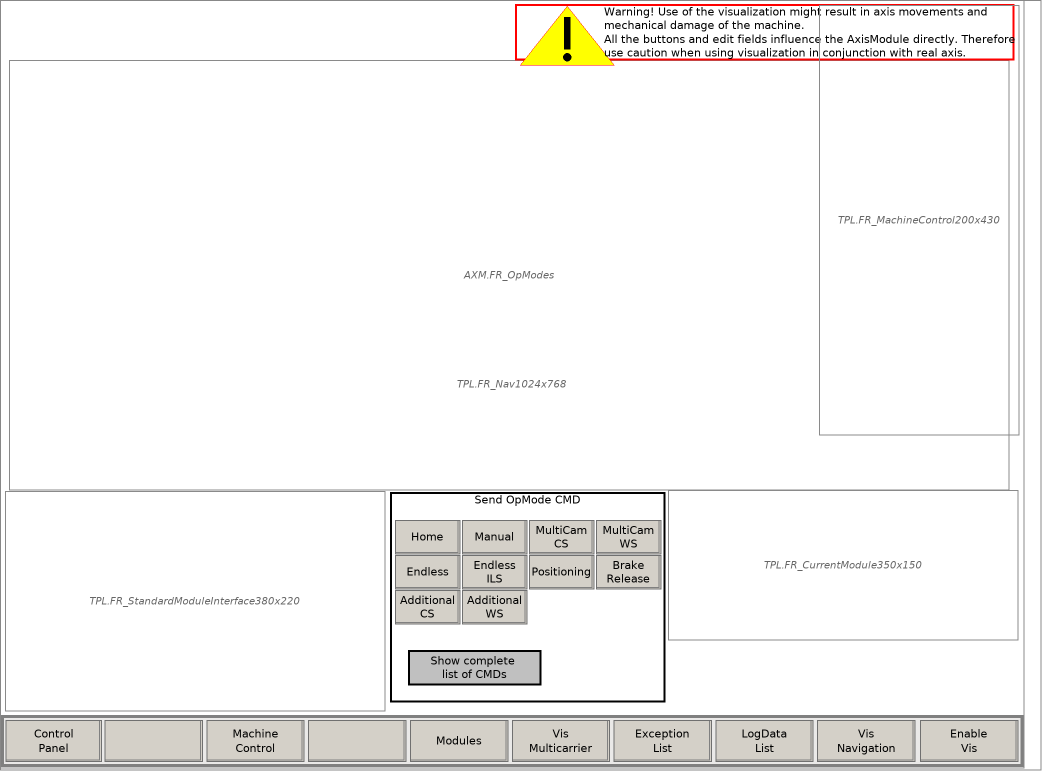
VISUALIZATION VIS_AxisModule  // 1042x771
    Frame (0,0 1024x768)
        shows TPL.FR_Nav1024x768(i_sTitle := 'Template: AxisModule')
    Frame (9,60 1000x430)
        shows AXM.FR_OpModes(iq_fbAxisModuleVisController := SR_VisControl.vpiq_fbAxisModuleVisController)
    Frame (5,491 380x220)
        shows TPL.FR_StandardModuleInterface380x220(i_stCurrentModuleStandardItf := SR_VisControl.vpq_stCurrentModuleStandardInterface, i_sCurrentModuleReaction := SR_VisControl.vpq_sCurrentModuleReaction, i_udiModuleReactionIndexMin := SR_VisControl.vpq_udiModuleReactionIndexMin, i_axModuleReaction := SR_VisControl.vpq_axModuleReaction, i_udiNumberOfReactions := SR_VisControl.udiCount, iq_xModuleReactionDown := SR_VisControl.vpiq_xModuleReactionDown, iq_xModuleReactionUp := SR_VisControl.vpiq_xModuleReactionUp, iq_diStartStepToSet := SR_VisControl.vpiq_diStartStepToSet, iq_diCmdToSet := SR_VisControl.vpiq_diCmdToSet, iq_xEnableModuleClicked := SR_VisControl.vpiq_xEnableModuleClicked, iq_xSetCmdClicked := SR_VisControl.vpiq_xSetCmdClicked, iq_fbVisContExHandling := SR_VisControl.vpiq_fbVisContExHandling)
    Rectangle (390,492 275x210), "Send OpMode CMD"
    Button (395,520 65x34), "Home", tooltip "Send CMD: ---------------------------------------------------------------- astSubModuleInterface[...].iq_diCMD := AXM.ET_Cmd.Homing (= 10);", colour toggle: SR_VisControl.v_xHomeModeActive, input disabled if: SR_VisControl.vpiq_fbAxisModuleVisController.i_pstCurrentStandardItf = 0
        OnMouseClick: execute { SR_VisControl.vpiq_fbAxisModuleVisController.i_pstCurrentStandardItf^.iq_diCmd := AXM.ET_Cmd.Homing; }
    Button (462,520 65x34), "Manual", tooltip "Send CMD: ---------------------------------------------------------------- astSubModuleInterface[...].iq_diCMD := AXM.ET_Cmd.Manual (= 20);", colour toggle: SR_VisControl.v_xManualModeActive, input disabled if: SR_VisControl.vpiq_fbAxisModuleVisController.i_pstCurrentStandardItf = 0
        OnMouseClick: execute { SR_VisControl.vpiq_fbAxisModuleVisController.i_pstCurrentStandardItf^.iq_diCmd := AXM.ET_Cmd.Manual; }
    Button (529,520 65x34), "MultiCam CS", tooltip "Send CMD: ---------------------------------------------------------------- astSubModuleInterface[...].iq_diCMD := AXM.ET_Cmd.CamCs (= 30);", colour toggle: SR_VisControl.v_xMultiCamCSActive, input disabled if: SR_VisControl.vpiq_fbAxisModuleVisController.i_pstCurrentStandardItf = 0
        OnMouseClick: execute { SR_VisControl.vpiq_fbAxisModuleVisController.i_pstCurrentStandardItf^.iq_diCmd := AXM.ET_Cmd.CamCs; }
    Button (596,520 65x34), "MultiCam WS", tooltip "Send CMD: ---------------------------------------------------------------- astSubModuleInterface[...].iq_diCMD := AXM.ET_Cmd.CamWs (= 31);", colour toggle: SR_VisControl.v_xMultiCamWSActive, input disabled if: SR_VisControl.vpiq_fbAxisModuleVisController.i_pstCurrentStandardItf = 0
        OnMouseClick: execute { SR_VisControl.vpiq_fbAxisModuleVisController.i_pstCurrentStandardItf^.iq_diCmd := AXM.ET_Cmd.CamWs; }
    Button (395,555 65x34), "Endless", tooltip "Send CMD: ---------------------------------------------------------------- astSubModuleInterface[...].iq_diCMD := AXM.ET_Cmd.Endless (= 40);", colour toggle: SR_VisControl.v_xEndlessActive, input disabled if: SR_VisControl.vpiq_fbAxisModuleVisController.i_pstCurrentStandardItf = 0
        OnMouseClick: execute { SR_VisControl.vpiq_fbAxisModuleVisController.i_pstCurrentStandardItf^.iq_diCmd := AXM.ET_Cmd.Endless; }
    Button (462,555 65x34), "Endless ILS", tooltip "Send CMD: ---------------------------------------------------------------- astSubModuleInterface[...].iq_diCMD := AXM.ET_Cmd.EndlessIls (= 41);", colour toggle: SR_VisControl.v_xEndlessILSActive, input disabled if: SR_VisControl.vpiq_fbAxisModuleVisController.i_pstCurrentStandardItf = 0
        OnMouseClick: execute { SR_VisControl.vpiq_fbAxisModuleVisController.i_pstCurrentStandardItf^.iq_diCmd := AXM.ET_Cmd.EndlessIls; }
    Button (529,555 65x34), "Positioning", tooltip "Send CMD: ---------------------------------------------------------------- astSubModuleInterface[...].iq_diCMD := AXM.ET_Cmd.Positioning (= 50);", colour toggle: SR_VisControl.v_xPositioningActive, input disabled if: SR_VisControl.vpiq_fbAxisModuleVisController.i_pstCurrentStandardItf = 0
        OnMouseClick: execute { SR_VisControl.vpiq_fbAxisModuleVisController.i_pstCurrentStandardItf^.iq_diCmd := AXM.ET_Cmd.Positioning; }
    Button (596,555 65x34), "Brake Release", tooltip "Send CMD: ---------------------------------------------------------------- astSubModuleInterface[...].iq_diCMD := AXM.ET_Cmd.BrakeRelease (= 70);", colour toggle: SR_VisControl.v_xBrakeActive, input disabled if: SR_VisControl.vpiq_fbAxisModuleVisController.i_pstCurrentStandardItf = 0
        OnMouseClick: execute { SR_VisControl.vpiq_fbAxisModuleVisController.i_pstCurrentStandardItf^.iq_diCmd := AXM.ET_Cmd.BrakeRelease; }
    Button (395,590 65x34), "Additional CS", tooltip "Send CMD: ---------------------------------------------------------------- astSubModuleInterface[...].iq_diCMD := AXM.ET_Cmd.AdditionalCs (= 80);", colour toggle: SR_VisControl.v_xAdditionalCSActive, input disabled if: SR_VisControl.vpiq_fbAxisModuleVisController.i_pstCurrentStandardItf = 0
        OnMouseClick: execute { SR_VisControl.vpiq_fbAxisModuleVisController.i_pstCurrentStandardItf^.iq_diCmd := AXM.ET_Cmd.AdditionalCs; }
    Button (462,590 65x34), "Additional WS", tooltip "Send CMD: ---------------------------------------------------------------- astSubModuleInterface[...].iq_diCMD := AXM.ET_Cmd.AdditionalWs (= 81);", colour toggle: SR_VisControl.v_xAdditionalWSActive, input disabled if: SR_VisControl.vpiq_fbAxisModuleVisController.i_pstCurrentStandardItf = 0
        OnMouseClick: execute { SR_VisControl.vpiq_fbAxisModuleVisController.i_pstCurrentStandardItf^.iq_diCmd := AXM.ET_Cmd.AdditionalWs; }
    Group (509,5 521x59)
        Rectangle (6,-1 499x56)
        Group (7,3 82x50)
            Polygon (4,57) (51,-2) (98,57) (98,57)
            Ellipse (47,45 8x8)
            RoundedRectangle (48,9 6x32)
        Rectangle (92,25 431x32), "All the buttons and edit fields influence the AxisModule directly. Therefore use caution when using visualization in conjunction with real axis."
        Rectangle (92,-2 439x31), "Warning! Use of the visualization might result in axis movements and mechanical damage of the machine."
    Frame (668,490 350x150)
        shows TPL.FR_CurrentModule350x150(i_stCurrentModuleStandardItf := SR_VisControl.vpq_stCurrentModuleStandardInterface)
    Rectangle (408,650 133x35), "Show complete list of CMDs", tooltip "(* AxisModule command area: 1-199 *) (*Selecting OpModes of FB_AxisModule*) Homing := 10 Manual := 20 CamCs := 30 CamWs := 31 Endless := 40 EndlessIls := 41 Positioning := 50 BrakeRelease := 70 AdditionalCs := 80 AdditionalWs := 81 (*ControlSignals for the selected OpMode of FB_AxisModule*) Start := 100 StartTrig := 101 StartTrigWaitInPos := 102 Stop := 110 Hold := 120 WsStart := 150 (*De-/Activating PositionControl of the respective Drive*) DriveEnableOn := 130 DriveEnableOff := 140"
    Frame (1,715 1024x54)
        shows FR_NavigationButtons()
    Frame (819,5 200x430), invisible if: NOT SR_VisControl.vpiq_xShowControlFrame
        shows TPL.FR_MachineControl200x430(i_stMachineItf := SR_VisControl.vpq_stMachineInterface, i_xPrepareActive := G_xPrepareActive, i_xAutoActive := G_xAutoActive, i_xBrakeReleaseActive := G_xBrakeReleaseActive, i_xJogMachineActive := G_xJogMachineActive, i_xManualActive := G_xManualActive, i_xException := SR_VisControl.vpq_xMachineInException, i_dwDiagQuitColor := SR_VisControl.vpq_dwDiagQuitColor, iq_iPositionX := SR_VisControl.vpiq_iPositionX, iq_iPositionY := SR_VisControl.vpiq_iPositionY, iq_xEmergencyEpas := G_xEmergencyEpas, iq_xStartEpas := G_xStartEpas, iq_xStopEpas := G_xStopEpas, iq_xJogForwEpas := G_xJogForwEpas, iq_xJogBackEpas := G_xJogBackEpas, iq_xDoPrepare := G_xDoPrepare, iq_xDoAuto := G_xDoAuto, iq_xDoBrakeRelease := G_xDoBrakeRelease, iq_xDoJogMachine := G_xDoJogMachine, iq_xDoManual := G_xDoManual, iq_xDiagQuitEpas := G_xDiagQuitEpas)
        p1457045297: SR_VisControl.stMachineInterface.stQ.xError
        p1941967854: g_I_xEmergency_Epas
        p2531571229: g_I_xStart_Epas
        p1511842254: g_I_xStop_Epas
        p745511063: g_I_xJogForw_Epas
        p3518271027: g_I_xJogBack_Epas
        p1982879521: g_I_xErrorQuit_Epas
        p3866886353: SR_VisControl.dwErrorQuitColor
        p1761348311: SR_VisControl.vpq_stMachineInterface
        p3560616238: SR_VisControl.vpiq_iPositionX
        p2738717112: SR_VisControl.vpiq_iPositionY
END_VISUALIZATION

// LMC_PacDrive/Application/TemplateFullProgrammingFramework/Visualization/Windows/VIS_ControlModule
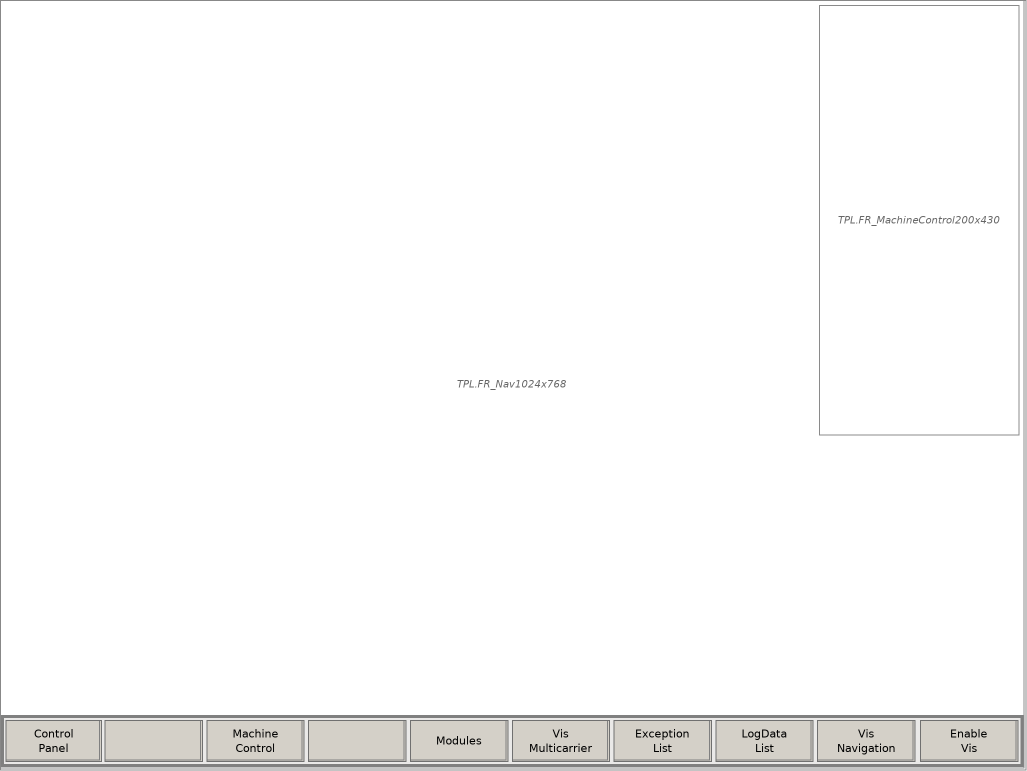
VISUALIZATION VIS_ControlModule  // 1027x771
    Frame (0,0 1024x768)
        shows TPL.FR_Nav1024x768(i_sTitle := 'Template: ControlModule')
    Frame (1,715 1024x54)
        shows FR_NavigationButtons()
    Frame (819,5 200x430), invisible if: NOT SR_VisControl.vpiq_xShowControlFrame
        shows TPL.FR_MachineControl200x430(i_stMachineItf := SR_VisControl.vpq_stMachineInterface, i_xPrepareActive := G_xPrepareActive, i_xAutoActive := G_xAutoActive, i_xBrakeReleaseActive := G_xBrakeReleaseActive, i_xJogMachineActive := G_xJogMachineActive, i_xManualActive := G_xManualActive, i_xException := SR_VisControl.vpq_xMachineInException, i_dwDiagQuitColor := SR_VisControl.vpq_dwDiagQuitColor, iq_iPositionX := SR_VisControl.vpiq_iPositionX, iq_iPositionY := SR_VisControl.vpiq_iPositionY, iq_xEmergencyEpas := G_xEmergencyEpas, iq_xStartEpas := G_xStartEpas, iq_xStopEpas := G_xStopEpas, iq_xJogForwEpas := G_xJogForwEpas, iq_xJogBackEpas := G_xJogBackEpas, iq_xDoPrepare := G_xDoPrepare, iq_xDoAuto := G_xDoAuto, iq_xDoBrakeRelease := G_xDoBrakeRelease, iq_xDoJogMachine := G_xDoJogMachine, iq_xDoManual := G_xDoManual, iq_xDiagQuitEpas := G_xDiagQuitEpas)
        p1457045297: SR_VisControl.stMachineInterface.stQ.xError
        p1941967854: g_I_xEmergency_Epas
        p2531571229: g_I_xStart_Epas
        p1511842254: g_I_xStop_Epas
        p745511063: g_I_xJogForw_Epas
        p3518271027: g_I_xJogBack_Epas
        p1982879521: g_I_xErrorQuit_Epas
        p3866886353: SR_VisControl.dwErrorQuitColor
        p1761348311: SR_VisControl.vpq_stMachineInterface
        p3560616238: SR_VisControl.vpiq_iPositionX
        p2738717112: SR_VisControl.vpiq_iPositionY
END_VISUALIZATION

// LMC_PacDrive/Application/TemplateFullProgrammingFramework/Visualization/Windows/VIS_ExceptionDetails
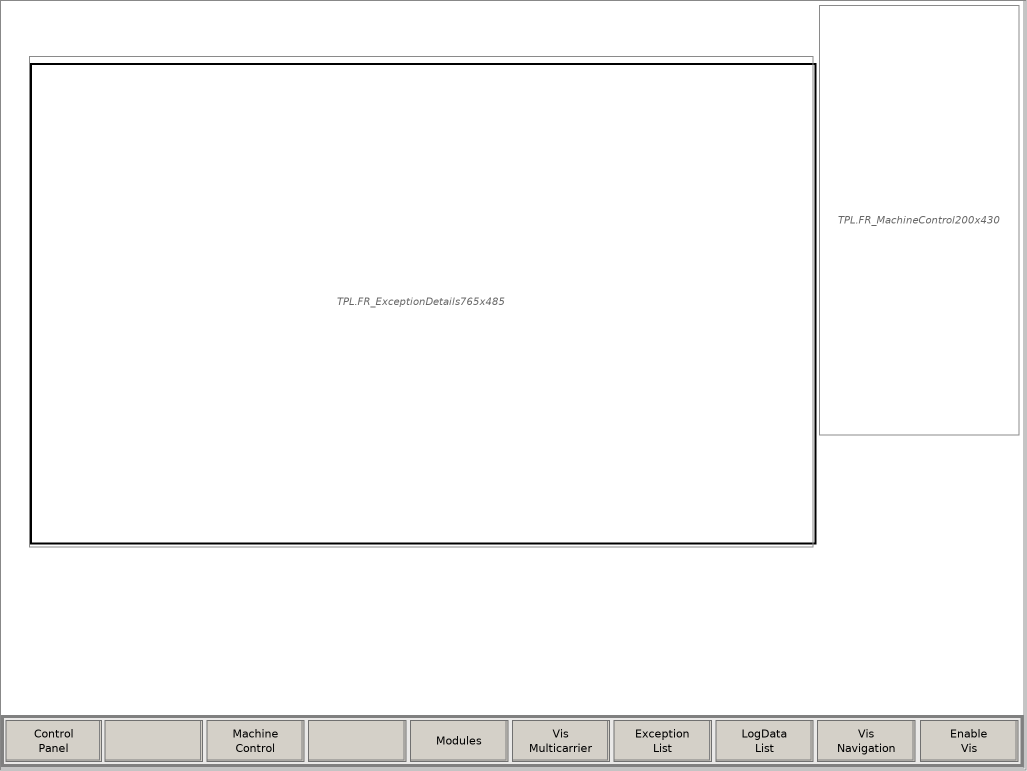
VISUALIZATION VIS_ExceptionDetails  // 1027x771
    Frame (0,0 1024x768)
        shows TPL.FR_Nav1024x768(i_sTitle := 'Template: ExceptionDetails')
    Frame (1,715 1024x54)
        shows FR_NavigationButtons()
    Rectangle (30,63 786x481)
    Frame (29,56 784x491)
        shows TPL.FR_ExceptionDetails765x485(iq_fbVisContExHandling := SR_VisControl.vpiq_fbVisContExHandling)
        p2566176161: 'Vis_ModuleErrors'
        p1989587566: 'Vis_Modules'
    Frame (819,5 200x430), invisible if: NOT SR_VisControl.vpiq_xShowControlFrame
        shows TPL.FR_MachineControl200x430(i_stMachineItf := SR_VisControl.vpq_stMachineInterface, i_xPrepareActive := G_xPrepareActive, i_xAutoActive := G_xAutoActive, i_xBrakeReleaseActive := G_xBrakeReleaseActive, i_xJogMachineActive := G_xJogMachineActive, i_xManualActive := G_xManualActive, i_xException := SR_VisControl.vpq_xMachineInException, i_dwDiagQuitColor := SR_VisControl.vpq_dwDiagQuitColor, iq_iPositionX := SR_VisControl.vpiq_iPositionX, iq_iPositionY := SR_VisControl.vpiq_iPositionY, iq_xEmergencyEpas := G_xEmergencyEpas, iq_xStartEpas := G_xStartEpas, iq_xStopEpas := G_xStopEpas, iq_xJogForwEpas := G_xJogForwEpas, iq_xJogBackEpas := G_xJogBackEpas, iq_xDoPrepare := G_xDoPrepare, iq_xDoAuto := G_xDoAuto, iq_xDoBrakeRelease := G_xDoBrakeRelease, iq_xDoJogMachine := G_xDoJogMachine, iq_xDoManual := G_xDoManual, iq_xDiagQuitEpas := G_xDiagQuitEpas)
        p1457045297: SR_VisControl.stMachineInterface.stQ.xError
        p1941967854: g_I_xEmergency_Epas
        p2531571229: g_I_xStart_Epas
        p1511842254: g_I_xStop_Epas
        p745511063: g_I_xJogForw_Epas
        p3518271027: g_I_xJogBack_Epas
        p1982879521: g_I_xErrorQuit_Epas
        p3866886353: SR_VisControl.dwErrorQuitColor
        p1761348311: SR_VisControl.vpq_stMachineInterface
        p3560616238: SR_VisControl.vpiq_iPositionX
        p2738717112: SR_VisControl.vpiq_iPositionY
END_VISUALIZATION

// LMC_PacDrive/Application/TemplateFullProgrammingFramework/Visualization/Windows/VIS_ExceptionList
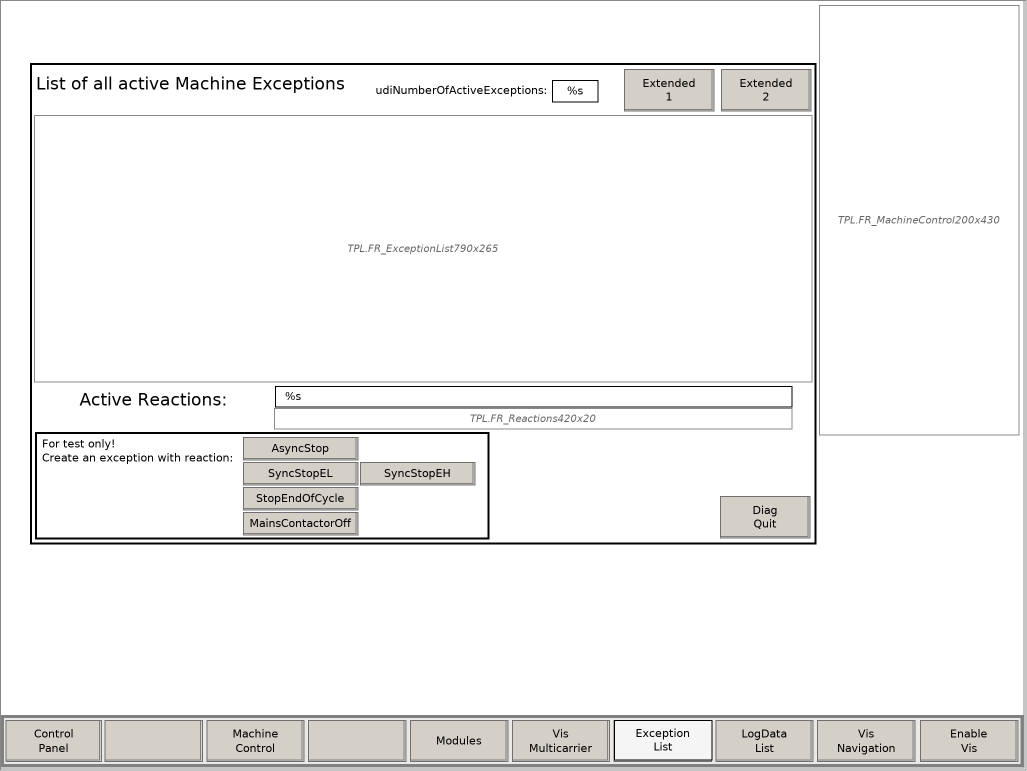
VISUALIZATION VIS_ExceptionList  // 1027x771
    Frame (0,0 1024x768)
        shows TPL.FR_Nav1024x768(i_sTitle := 'Template: ExceptionList')
    Frame (1,715 1024x54)
        shows FR_NavigationButtons()
    Rectangle (30,63 786x481)
    Rectangle (33,66 310x35), "List of all active Machine Exceptions"
    Rectangle (46,382 215x35), "Active Reactions:"
    Rectangle (369,78 181x25), "udiNumberOfActiveExceptions:"
    Rectangle (275,386 517x21), "%s", text variable: SR_VisControl.vpq_sAllActiveReactions
    Rectangle (35,432 454x107)
    Rectangle (39,436 195x29), "For test only! Create an exception with reaction:"
    Frame (274,408 518x21)
        shows TPL.FR_Reactions420x20(i_udiIndexMin := SR_VisControl.vpq_udiReactionIndexMin, i_axReaction := SR_VisControl.vpq_axReaction, i_udiNumberOfReactions := TPL.Gc_udiMaxNumberOfReactions, iq_xScrollDown := SR_VisControl.vpiq_xReactionDown, iq_xScrollUp := SR_VisControl.vpiq_xReactionUp)
        p3944911060: SR_VisControl.iErrorReactionIndexMin
        p214250784: TPC_Gc_diMaxNumberOfErrorReactions
    Button (360,462 115x23), "SyncStopEH", tooltip "For testing purpose only! Create an exception with the reaction TPL.ET_Reaction.SyncStopEH. Machine reacts with "Synchronous stop". For a detailed description of this reaction search the help index for ET_Reaction.", colour toggle: SR_VisControl.vpiq_xTestUserException3
        toggle SR_VisControl.vpiq_xTestUserException3
    Button (243,437 115x23), "AsyncStop", tooltip "For testing purpose only! Create an exception with the reaction TPL.ET_Reaction.AsyncStop. Machine reacts with "Immediate asynchronous stop". For a detailed description of this reaction search the help index for ET_Reaction.", colour toggle: SR_VisControl.vpiq_xTestUserException1
        toggle SR_VisControl.vpiq_xTestUserException1
    Button (243,462 115x23), "SyncStopEL", tooltip "For testing purpose only! Create an exception with the reaction TPL.ET_Reaction.SyncStopEL. Machine reacts with "Synchronous stop with process deactivation after stop". For a detailed description of this reaction search the help index for ET_Reaction.", colour toggle: SR_VisControl.vpiq_xTestUserException2
        toggle SR_VisControl.vpiq_xTestUserException2
    Button (243,487 115x23), "StopEndOfCycle", tooltip "For testing purpose only! Create an exception with the reaction TPL.ET_Reaction.StopEndOfCycle. Machine reacts with "Stop at end of cycle". For a detailed description of this reaction search the help index for ET_Reaction.", colour toggle: SR_VisControl.vpiq_xTestUserException4
        toggle SR_VisControl.vpiq_xTestUserException4
    Button (243,512 115x23), "MainsContactorOff", tooltip "For testing purpose only! Create an exception with the reaction TPL.ET_Reaction.MainsContactorOff. Machine reacts with "Immediate deactivation of the mains contactor". For a detailed description of this reaction search the help index for ET_Reaction.", colour toggle: SR_VisControl.vpiq_xTestUserException5
        toggle SR_VisControl.vpiq_xTestUserException5
    Button (624,69 90x42), "Extended 1", colour toggle: SR_VisControl.vpq_xShowExtendedTimes
        toggle SR_VisControl.vpiq_xButtonShowExtendedTimes
    Button (721,69 90x42), "Extended 2", colour toggle: SR_VisControl.vpq_xShowExtended2
        toggle SR_VisControl.vpiq_xButtonShowExtended2
    Textfield (552,80 46x22), "%s", text variable: G_stExceptionList.udiNumberOfActiveExceptions
    Button (720,496 90x42), "Diag Quit", colour toggle: SR_VisControl.vpq_xMachineInException
        p573394764: SR_VisControl.vpq_dwDiagQuitColor
        tap G_xDiagQuitEpas
    Frame (34,115 778x267)
        shows TPL.FR_ExceptionList790x265(i_astExceptionListTable := SR_VisControl.vpq_astExceptionListTable, i_asReaction := SR_VisControl.vpq_asReaction, i_xShowExtendedTimes := SR_VisControl.vpq_xShowExtendedTimes, i_xShowExtended2 := SR_VisControl.vpq_xShowExtended2, i_xDisplayScrollDown := SR_VisControl.vpq_xDisplayScrollDown, i_udiExceptionListIndexMax := SR_VisControl.vpq_udiExceptionListIndexMax, i_udiNumberOfExceptions := SR_VisControl.vpq_udiNumberOfExceptions, iq_udiExceptionListIndexMin := SR_VisControl.vpiq_udiExceptionListIndexMin, iq_udiExceptionListGoToDetailsOfLine := SR_VisControl.vpiq_udiExceptionListGoToDetailsOfLine)
    Rectangle (614,720 98x40), "Exception List"
    Frame (819,5 200x430), invisible if: NOT SR_VisControl.vpiq_xShowControlFrame
        shows TPL.FR_MachineControl200x430(i_stMachineItf := SR_VisControl.vpq_stMachineInterface, i_xPrepareActive := G_xPrepareActive, i_xAutoActive := G_xAutoActive, i_xBrakeReleaseActive := G_xBrakeReleaseActive, i_xJogMachineActive := G_xJogMachineActive, i_xManualActive := G_xManualActive, i_xException := SR_VisControl.vpq_xMachineInException, i_dwDiagQuitColor := SR_VisControl.vpq_dwDiagQuitColor, iq_iPositionX := SR_VisControl.vpiq_iPositionX, iq_iPositionY := SR_VisControl.vpiq_iPositionY, iq_xEmergencyEpas := G_xEmergencyEpas, iq_xStartEpas := G_xStartEpas, iq_xStopEpas := G_xStopEpas, iq_xJogForwEpas := G_xJogForwEpas, iq_xJogBackEpas := G_xJogBackEpas, iq_xDoPrepare := G_xDoPrepare, iq_xDoAuto := G_xDoAuto, iq_xDoBrakeRelease := G_xDoBrakeRelease, iq_xDoJogMachine := G_xDoJogMachine, iq_xDoManual := G_xDoManual, iq_xDiagQuitEpas := G_xDiagQuitEpas)
        p1457045297: SR_VisControl.stMachineInterface.stQ.xError
        p1941967854: g_I_xEmergency_Epas
        p2531571229: g_I_xStart_Epas
        p1511842254: g_I_xStop_Epas
        p745511063: g_I_xJogForw_Epas
        p3518271027: g_I_xJogBack_Epas
        p1982879521: g_I_xErrorQuit_Epas
        p3866886353: SR_VisControl.dwErrorQuitColor
        p1761348311: SR_VisControl.vpq_stMachineInterface
        p3560616238: SR_VisControl.vpiq_iPositionX
        p2738717112: SR_VisControl.vpiq_iPositionY
END_VISUALIZATION

// LMC_PacDrive/Application/TemplateFullProgrammingFramework/Visualization/Windows/VIS_LogDataList
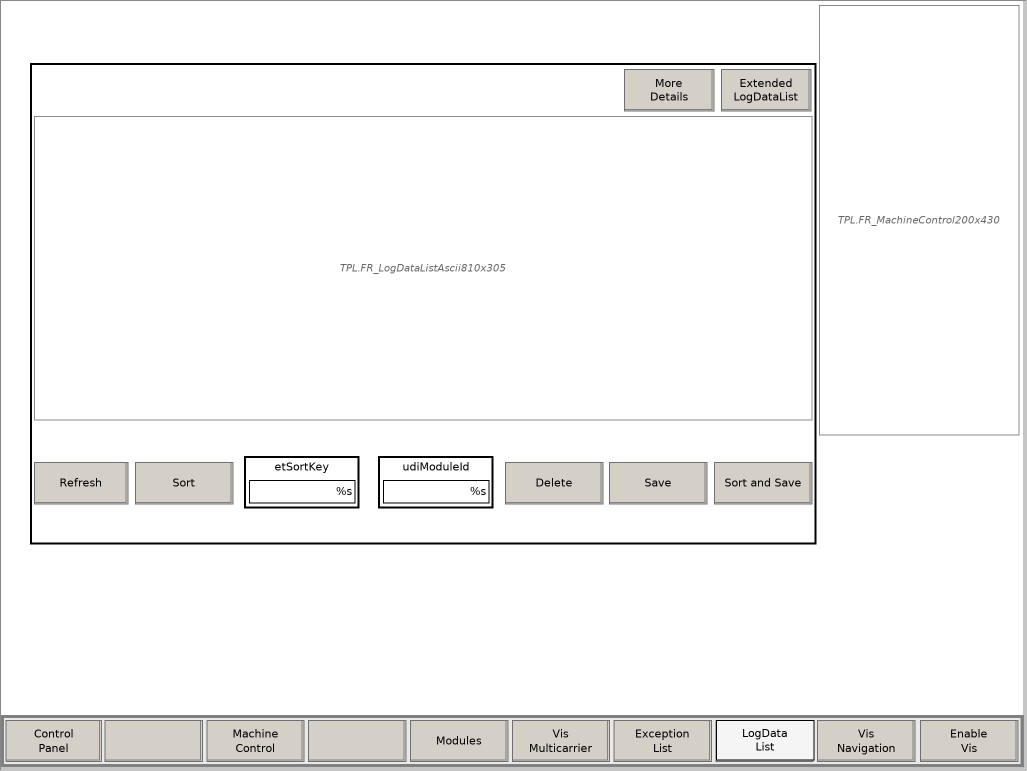
VISUALIZATION VIS_LogDataList  // 1027x771
    Frame (0,0 1024x768)
        shows TPL.FR_Nav1024x768(i_sTitle := 'Template: LogDataList')
    Frame (1,715 1024x54)
        shows FR_NavigationButtons()
    Rectangle (30,63 786x481)
    Rectangle (244,456 115x52)
    Rectangle (378,456 115x52)
    Frame (34,116 778x304)
        shows TPL.FR_LogDataListAscii810x305(i_udiLogDataListIndexMax := SR_VisControl.vpq_udiLogDataListIndexMax, i_xLogDataScrollDown := SR_VisControl.vpq_xLogDataScrollDown, i_stLogDataListAscii := G_stLogDataListAscii, i_astLogDataTable := SR_VisControl.vpq_astLogDataTable, i_xShowLogDataListDetails := SR_VisControl.vpq_xShowLogDataListDetails, iq_udiLogDataListIndexMin := SR_VisControl.vpiq_udiLogDataListIndexMin, iq_udiNumberOfLogData := SR_VisControl.vpiq_udiNumberOfLogData)
        p614390240: SR_VisControl.iLoggerListIndexMin
        p2848728500: G_stLogDataListAscii
        p1478497087: SR_VisControl.xLoggerExtendedLogger
        p3640196843: SR_VisControl.xLoggerScrollDown
        p3171618909: SR_VisControl.diNumberOfLogData
        p348598905: SR_VisControl.iLoggerListIndexMax
        p443021939: SR_VisControl.udiLoggerListIndexMax
        p1814956285: SR_VisControl.udiLoggerListIndexMin
    Button (624,69 90x42), "More Details", colour toggle: SR_VisControl.vpq_xShowLogDataListDetails
        toggle SR_VisControl.vpiq_xButtonLogDataListDetails
    Button (721,69 90x42), "Extended LogDataList"
        OnMouseClick:  Assign=VIS_LogDataListExt, Type=Assignment
    Button (135,462 98x42), "Sort", colour toggle: G_stLoggerInterface.i_xSort
        tap G_stLoggerInterface.i_xSort
    Button (34,462 94x42), "Refresh", colour toggle: G_stLoggerInterface.i_xSort
        tap G_stLoggerInterface.i_xSort
    Button (505,462 98x42), "Delete", colour toggle: G_stLoggerInterface.i_xDelete
        tap G_stLoggerInterface.i_xDelete
    Button (609,462 98x42), "Save", colour toggle: G_stLoggerInterface.i_xSave
        tap G_stLoggerInterface.i_xSave
    Button (714,462 98x42), "Sort and Save", colour toggle: G_stLoggerInterface.i_xSortAndSave
        tap G_stLoggerInterface.i_xSortAndSave
    Textfield (383,480 106x23), "%s", text variable: G_stLoggerInterface.i_udiModuleId
        OnMouseClick: write the text variable via Edit
    Textfield (249,480 106x23), "%s", tooltip "TPD_SORTBY_TIME:= 0 TPD_SORTBY_NAME:= 1 TPD_SORTBY_ID:= 2 TPD_SORTBY_CMD:= 3 TPD_SORTBY_ERRORREACTION:= 4 TPD_GE_SORTBY_MODULE_ID:= 5 TPD_GE_SORTBY_MODULE_ID_AND_TIME:= 6", text variable: G_stLoggerInterface.i_etSortKey
        OnMouseClick: write the text variable via Edit
    Rectangle (247,458 110x18), "etSortKey"
    Rectangle (381,458 110x18), "udiModuleId"
    Rectangle (716,720 98x40), "LogData List"
    Frame (819,5 200x430), invisible if: NOT SR_VisControl.vpiq_xShowControlFrame
        shows TPL.FR_MachineControl200x430(i_stMachineItf := SR_VisControl.vpq_stMachineInterface, i_xPrepareActive := G_xPrepareActive, i_xAutoActive := G_xAutoActive, i_xBrakeReleaseActive := G_xBrakeReleaseActive, i_xJogMachineActive := G_xJogMachineActive, i_xManualActive := G_xManualActive, i_xException := SR_VisControl.vpq_xMachineInException, i_dwDiagQuitColor := SR_VisControl.vpq_dwDiagQuitColor, iq_iPositionX := SR_VisControl.vpiq_iPositionX, iq_iPositionY := SR_VisControl.vpiq_iPositionY, iq_xEmergencyEpas := G_xEmergencyEpas, iq_xStartEpas := G_xStartEpas, iq_xStopEpas := G_xStopEpas, iq_xJogForwEpas := G_xJogForwEpas, iq_xJogBackEpas := G_xJogBackEpas, iq_xDoPrepare := G_xDoPrepare, iq_xDoAuto := G_xDoAuto, iq_xDoBrakeRelease := G_xDoBrakeRelease, iq_xDoJogMachine := G_xDoJogMachine, iq_xDoManual := G_xDoManual, iq_xDiagQuitEpas := G_xDiagQuitEpas)
        p1457045297: SR_VisControl.stMachineInterface.stQ.xError
        p1941967854: g_I_xEmergency_Epas
        p2531571229: g_I_xStart_Epas
        p1511842254: g_I_xStop_Epas
        p745511063: g_I_xJogForw_Epas
        p3518271027: g_I_xJogBack_Epas
        p1982879521: g_I_xErrorQuit_Epas
        p3866886353: SR_VisControl.dwErrorQuitColor
        p1761348311: SR_VisControl.vpq_stMachineInterface
        p3560616238: SR_VisControl.vpiq_iPositionX
        p2738717112: SR_VisControl.vpiq_iPositionY
END_VISUALIZATION

// LMC_PacDrive/Application/TemplateFullProgrammingFramework/Visualization/Windows/VIS_LogDataListExt
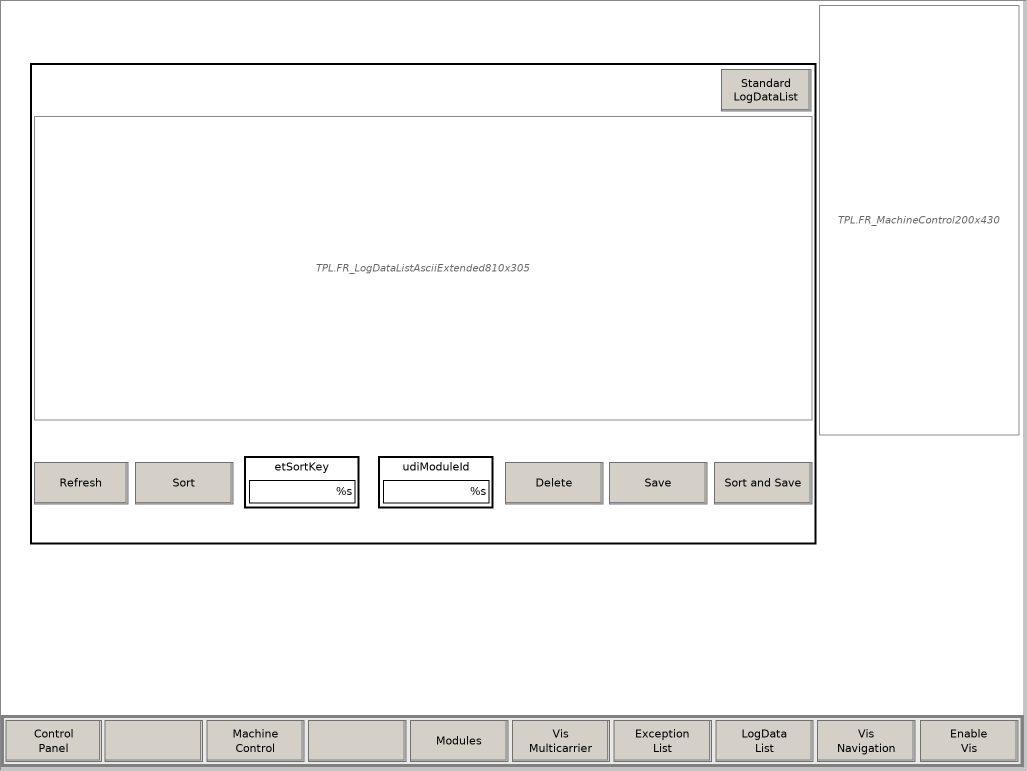
VISUALIZATION VIS_LogDataListExt  // 1027x771
    Frame (0,0 1024x768)
        shows TPL.FR_Nav1024x768(i_sTitle := 'Template: LogDataListExt')
    Frame (1,715 1024x54)
        shows FR_NavigationButtons()
    Rectangle (30,63 786x481)
    Rectangle (244,456 115x52)
    Rectangle (378,456 115x52)
    Button (135,462 98x42), "Sort", colour toggle: G_stLoggerInterface.i_xSort
        tap G_stLoggerInterface.i_xSort
    Button (34,462 94x42), "Refresh", colour toggle: G_stLoggerInterface.i_xSort
        tap G_stLoggerInterface.i_xSort
    Button (505,462 98x42), "Delete", colour toggle: G_stLoggerInterface.i_xDelete
        tap G_stLoggerInterface.i_xDelete
    Button (609,462 98x42), "Save", colour toggle: G_stLoggerInterface.i_xSave
        tap G_stLoggerInterface.i_xSave
    Button (714,462 98x42), "Sort and Save", colour toggle: G_stLoggerInterface.i_xSortAndSave
        tap G_stLoggerInterface.i_xSortAndSave
    Textfield (383,480 106x23), "%s", text variable: G_stLoggerInterface.i_udiModuleId
        OnMouseClick: write the text variable via Edit
    Textfield (249,480 106x23), "%s", tooltip "TPD_SORTBY_TIME:= 0 TPD_SORTBY_NAME:= 1 TPD_SORTBY_ID:= 2 TPD_SORTBY_CMD:= 3 TPD_SORTBY_ERRORREACTION:= 4 TPD_GE_SORTBY_MODULE_ID:= 5 TPD_GE_SORTBY_MODULE_ID_AND_TIME:= 6", text variable: G_stLoggerInterface.i_etSortKey
        OnMouseClick: write the text variable via Edit
    Rectangle (247,458 110x18), "etSortKey"
    Rectangle (381,458 110x18), "udiModuleId"
    Button (721,69 90x42), "Standard LogDataList"
        OnMouseClick:  Assign=VIS_LogDataList, Type=Assignment
    Frame (34,116 778x304)
        shows TPL.FR_LogDataListAsciiExtended810x305(i_udiLogDataListIndexMax := SR_VisControl.vpq_udiLogDataListIndexMax, i_xLogDataScrollDown := SR_VisControl.vpq_xLogDataScrollDown, i_stLogDataListAscii := G_stLogDataListAscii, i_astLogDataTable := SR_VisControl.vpq_astLogDataTable, i_astLogDataTableAscii := SR_VisControl.vpq_astLogDataTableAscii, iq_udiLogDataListIndexMin := SR_VisControl.vpiq_udiLogDataListIndexMin, iq_udiNumberOfLogData := SR_VisControl.vpiq_udiNumberOfLogData)
        p2848728500: G_stLogDataListAscii
        p3166277772: SR_VisControl.astLogDataTable
        p348598905: SR_VisControl.iLoggerListIndexMax
        p614390240: SR_VisControl.iLoggerListIndexMin
        p3640196843: SR_VisControl.xLoggerScrollDown
        p3171618909: SR_VisControl.diNumberOfLogData
        p443021939: SR_VisControl.udiLoggerListIndexMax
        p1478497087: SR_VisControl.xLoggerExtendedLogger
        p1814956285: SR_VisControl.udiLoggerListIndexMin
    Frame (819,5 200x430), invisible if: NOT SR_VisControl.vpiq_xShowControlFrame
        shows TPL.FR_MachineControl200x430(i_stMachineItf := SR_VisControl.vpq_stMachineInterface, i_xPrepareActive := G_xPrepareActive, i_xAutoActive := G_xAutoActive, i_xBrakeReleaseActive := G_xBrakeReleaseActive, i_xJogMachineActive := G_xJogMachineActive, i_xManualActive := G_xManualActive, i_xException := SR_VisControl.vpq_xMachineInException, i_dwDiagQuitColor := SR_VisControl.vpq_dwDiagQuitColor, iq_iPositionX := SR_VisControl.vpiq_iPositionX, iq_iPositionY := SR_VisControl.vpiq_iPositionY, iq_xEmergencyEpas := G_xEmergencyEpas, iq_xStartEpas := G_xStartEpas, iq_xStopEpas := G_xStopEpas, iq_xJogForwEpas := G_xJogForwEpas, iq_xJogBackEpas := G_xJogBackEpas, iq_xDoPrepare := G_xDoPrepare, iq_xDoAuto := G_xDoAuto, iq_xDoBrakeRelease := G_xDoBrakeRelease, iq_xDoJogMachine := G_xDoJogMachine, iq_xDoManual := G_xDoManual, iq_xDiagQuitEpas := G_xDiagQuitEpas)
        p1457045297: SR_VisControl.stMachineInterface.stQ.xError
        p1941967854: g_I_xEmergency_Epas
        p2531571229: g_I_xStart_Epas
        p1511842254: g_I_xStop_Epas
        p745511063: g_I_xJogForw_Epas
        p3518271027: g_I_xJogBack_Epas
        p1982879521: g_I_xErrorQuit_Epas
        p3866886353: SR_VisControl.dwErrorQuitColor
        p1761348311: SR_VisControl.vpq_stMachineInterface
        p3560616238: SR_VisControl.vpiq_iPositionX
        p2738717112: SR_VisControl.vpiq_iPositionY
END_VISUALIZATION

// LMC_PacDrive/Application/TemplateFullProgrammingFramework/Visualization/Windows/VIS_ModuleDetails
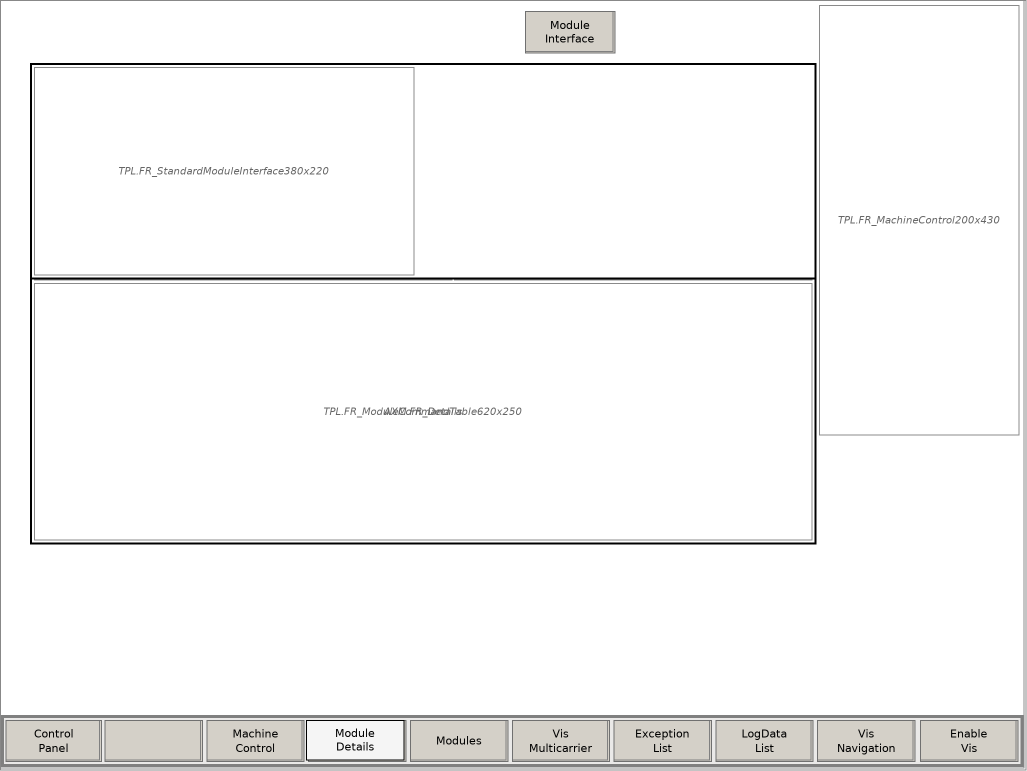
VISUALIZATION VIS_ModuleDetails  // 1027x771
    Frame (0,0 1024x768)
        shows TPL.FR_Nav1024x768(i_sTitle := 'Template: ModuleDetails')
    Frame (1,715 1024x54)
        shows FR_NavigationButtons()
    Button (525,11 90x42), "Module Interface", colour toggle: SR_VisControl.vpiq_xShowModuleInterface
        toggle SR_VisControl.vpiq_xShowModuleInterface
    Rectangle (30,63 786x481)
    Frame (34,128 418x152)
        shows TPL.FR_Navigation360x150(i_sNameNavRight := SR_VisControl.vpq_sNameNavRight, i_sNameNavUp := SR_VisControl.vpq_sNameNavUp, i_sNameNavLeft := SR_VisControl.vpq_sNameNavLeft, i_sNameNavDown := SR_VisControl.vpq_sNameNavDown, i_xEnableNavUp := SR_VisControl.vpq_xEnableNavUp, i_xEnableNavLeft := SR_VisControl.vpq_xEnableNavLeft, i_xEnableNavRight := SR_VisControl.vpq_xEnableNavRight, i_xEnableNavDown := SR_VisControl.vpq_xEnableNavDown, iq_xNavUp := SR_VisControl.vpiq_xNavUp, iq_xNavLeft := SR_VisControl.vpiq_xNavLeft, iq_xNavRight := SR_VisControl.vpiq_xNavRight, iq_xNavDown := SR_VisControl.vpiq_xNavDown)
    Rectangle (30,64 786x60)
    Button (602,65 118x29), "EQModule: %s", tooltip "%s", text variable: SR_VisControl.vpq_audiIdModuleList[5], colour toggle: SR_VisControl.vpq_axActiveModuleList[5], invisible if: SR_VisControl.vpq_axDisableModuleList[5] OR SR_VisControl.vpq_axIdModuleListValid[5] = FALSE, input disabled if: SR_VisControl.vpq_axDisableModuleList[5]
        p4168582468: SR_VisControl.vpq_asNameModuleList[5]
        toggle SR_VisControl.vpiq_axModuleList[5]
    Button (483,65 118x29), "EQModule: %s", tooltip "%s", text variable: SR_VisControl.vpq_audiIdModuleList[4], colour toggle: SR_VisControl.vpq_axActiveModuleList[4], invisible if: SR_VisControl.vpq_axDisableModuleList[4] OR SR_VisControl.vpq_axIdModuleListValid[4] = FALSE, input disabled if: SR_VisControl.vpq_axDisableModuleList[4]
        p4168582468: SR_VisControl.vpq_asNameModuleList[4]
        toggle SR_VisControl.vpiq_axModuleList[4]
    Button (365,65 118x29), "EQModule: %s", tooltip "%s", text variable: SR_VisControl.vpq_audiIdModuleList[3], colour toggle: SR_VisControl.vpq_axActiveModuleList[3], invisible if: SR_VisControl.vpq_axDisableModuleList[3] OR SR_VisControl.vpq_axIdModuleListValid[3] = FALSE, input disabled if: SR_VisControl.vpq_axDisableModuleList[3]
        p4168582468: SR_VisControl.vpq_asNameModuleList[3]
        toggle SR_VisControl.vpiq_axModuleList[3]
    Button (246,65 118x29), "EQModule: %s", tooltip "%s", text variable: SR_VisControl.vpq_audiIdModuleList[2], colour toggle: SR_VisControl.vpq_axActiveModuleList[2], invisible if: SR_VisControl.vpq_axDisableModuleList[2] OR SR_VisControl.vpq_axIdModuleListValid[2] = FALSE, input disabled if: SR_VisControl.vpq_axDisableModuleList[2]
        p4168582468: SR_VisControl.vpq_asNameModuleList[2]
        toggle SR_VisControl.vpiq_axModuleList[2]
    Button (126,65 119x29), "EQModule: %s", tooltip "%s", text variable: SR_VisControl.vpq_audiIdModuleList[1], colour toggle: SR_VisControl.vpq_axActiveModuleList[1], invisible if: SR_VisControl.vpq_axDisableModuleList[1] OR SR_VisControl.vpq_axIdModuleListValid[1] = FALSE, input disabled if: SR_VisControl.vpq_axDisableModuleList[1]
        p4168582468: SR_VisControl.vpq_asNameModuleList[1]
        toggle SR_VisControl.vpiq_axModuleList[1]
    Button (126,95 119x29), "SubEQModule: %s", tooltip "%s", text variable: SR_VisControl.vpq_audiIdSubModuleList[1], colour toggle: SR_VisControl.vpq_axActiveSubModuleList[1], invisible if: SR_VisControl.vpq_axDisableSubModuleList[1] OR SR_VisControl.vpq_axIdSubModuleListValid[1] = FALSE, input disabled if: SR_VisControl.vpq_axDisableSubModuleList[1]
        p4168582468: SR_VisControl.vpq_asNameSubModuleList[1]
        toggle SR_VisControl.vpiq_axSubModuleList[1]
    Button (246,95 118x29), "SubEQModule: %s", tooltip "%s", text variable: SR_VisControl.vpq_audiIdSubModuleList[2], colour toggle: SR_VisControl.vpq_axActiveSubModuleList[2], invisible if: SR_VisControl.vpq_axDisableSubModuleList[2] OR SR_VisControl.vpq_axIdSubModuleListValid[2] = FALSE, input disabled if: SR_VisControl.vpq_axDisableSubModuleList[2]
        p4168582468: SR_VisControl.vpq_asNameSubModuleList[2]
        toggle SR_VisControl.vpiq_axSubModuleList[2]
    Button (365,95 118x29), "SubEQModule: %s", tooltip "%s", text variable: SR_VisControl.vpq_audiIdSubModuleList[3], colour toggle: SR_VisControl.vpq_axActiveSubModuleList[3], invisible if: SR_VisControl.vpq_axDisableSubModuleList[3] OR SR_VisControl.vpq_axIdSubModuleListValid[3] = FALSE, input disabled if: SR_VisControl.vpq_axDisableSubModuleList[3]
        p4168582468: SR_VisControl.vpq_asNameSubModuleList[3]
        toggle SR_VisControl.vpiq_axSubModuleList[3]
    Button (484,95 117x29), "SubEQModule: %s", tooltip "%s", text variable: SR_VisControl.vpq_audiIdSubModuleList[4], colour toggle: SR_VisControl.vpq_axActiveSubModuleList[4], invisible if: SR_VisControl.vpq_axDisableSubModuleList[4] OR SR_VisControl.vpq_axIdSubModuleListValid[4] = FALSE, input disabled if: SR_VisControl.vpq_axDisableSubModuleList[4]
        p4168582468: SR_VisControl.vpq_asNameSubModuleList[4]
        toggle SR_VisControl.vpiq_axSubModuleList[4]
    Button (602,95 118x29), "SubEQModule: %s", tooltip "%s", text variable: SR_VisControl.vpq_audiIdSubModuleList[5], colour toggle: SR_VisControl.vpq_axActiveSubModuleList[5], invisible if: SR_VisControl.vpq_axDisableSubModuleList[5] OR SR_VisControl.vpq_axIdSubModuleListValid[5] = FALSE, input disabled if: SR_VisControl.vpq_axDisableSubModuleList[5]
        p4168582468: SR_VisControl.vpq_asNameSubModuleList[5]
        toggle SR_VisControl.vpiq_axSubModuleList[5]
    Rectangle (720,94 95x29), ">"
    Rectangle (720,64 95x30), ">"
    Button (721,65 95x29), ">", invisible if: SR_VisControl.vpq_xDisableModuleListUp, input disabled if: SR_VisControl.vpq_xDisableModuleListUp
        toggle SR_VisControl.vpiq_xModuleListUp
    Button (721,95 95x29), ">", invisible if: SR_VisControl.vpq_xDisableSubModuleListUp, input disabled if: SR_VisControl.vpq_xDisableSubModuleListUp
        toggle SR_VisControl.vpiq_xSubModuleListUp
    Rectangle (31,94 94x29), "<"
    Rectangle (31,64 94x30), "<"
    Button (32,65 93x29), "<", invisible if: SR_VisControl.vpq_xDisableModuleListDown, input disabled if: SR_VisControl.vpq_xDisableModuleListDown
        toggle SR_VisControl.vpiq_xModuleListDown
    Button (32,95 93x29), "<", invisible if: SR_VisControl.vpq_xDisableSubModuleListDown, input disabled if: SR_VisControl.vpq_xDisableSubModuleListDown
        toggle SR_VisControl.vpiq_xSubModuleListDown
    Button (126,65 119x29), "CtrlModule: %s", tooltip "%s", text variable: SR_VisControl.vpq_asControlModuleButtonName[1], colour toggle: SR_VisControl.vpq_axControlModuleActive[1], invisible if: SR_VisControl.vpq_axControlModuleValid[1]=FALSE
        p4168582468: SR_VisControl.vpq_asToolTipControlModuleList[1]
        toggle SR_VisControl.vpiq_axControlModuleList[1]
    Button (246,65 118x29), "CtrlModule: %s", tooltip "%s", text variable: SR_VisControl.vpq_asControlModuleButtonName[2], colour toggle: SR_VisControl.vpq_axControlModuleActive[2], invisible if: SR_VisControl.vpq_axControlModuleValid[2]=FALSE
        p4168582468: SR_VisControl.vpq_asToolTipControlModuleList[2]
        toggle SR_VisControl.vpiq_axControlModuleList[2]
    Button (365,65 118x29), "CtrlModule: %s", tooltip "%s", text variable: SR_VisControl.vpq_asControlModuleButtonName[3], colour toggle: SR_VisControl.vpq_axControlModuleActive[3], invisible if: SR_VisControl.vpq_axControlModuleValid[3]=FALSE
        p4168582468: SR_VisControl.vpq_asToolTipControlModuleList[3]
        toggle SR_VisControl.vpiq_axControlModuleList[3]
    Button (484,65 117x29), "CtrlModule: %s", tooltip "%s", text variable: SR_VisControl.vpq_asControlModuleButtonName[4], colour toggle: SR_VisControl.vpq_axControlModuleActive[4], invisible if: SR_VisControl.vpq_axControlModuleValid[4]=FALSE
        p4168582468: SR_VisControl.vpq_asToolTipControlModuleList[4]
        toggle SR_VisControl.vpiq_axControlModuleList[4]
    Button (602,65 118x29), "CtrlModule: %s", tooltip "%s", text variable: SR_VisControl.vpq_asControlModuleButtonName[5], colour toggle: SR_VisControl.vpq_axControlModuleActive[5], invisible if: SR_VisControl.vpq_axControlModuleValid[5]=FALSE
        p4168582468: SR_VisControl.vpq_asToolTipControlModuleList[5]
        toggle SR_VisControl.vpiq_axControlModuleList[5]
    Button (126,95 119x29), "SubCtrlModule: %s", tooltip "%s", text variable: SR_VisControl.vpq_asSubControlModuleButtonName[1], colour toggle: SR_VisControl.vpq_axSubControlModuleActive[1], invisible if: SR_VisControl.vpq_axSubControlModuleValid[1]=FALSE
        p4168582468: SR_VisControl.vpq_asToolTipSubControlModuleList[1]
        toggle SR_VisControl.vpiq_axSubControlModuleList[1]
    Button (246,95 118x29), "SubCtrlModule: %s", tooltip "%s", text variable: SR_VisControl.vpq_asSubControlModuleButtonName[2], colour toggle: SR_VisControl.vpq_axSubControlModuleActive[2], invisible if: SR_VisControl.vpq_axSubControlModuleValid[2]=FALSE
        p4168582468: SR_VisControl.vpq_asToolTipSubControlModuleList[2]
        toggle SR_VisControl.vpiq_axSubControlModuleList[2]
    Button (365,95 118x29), "SubCtrlModule: %s", tooltip "%s", text variable: SR_VisControl.vpq_asSubControlModuleButtonName[3], colour toggle: SR_VisControl.vpq_axSubControlModuleActive[3], invisible if: SR_VisControl.vpq_axSubControlModuleValid[3]=FALSE
        p4168582468: SR_VisControl.vpq_asToolTipSubControlModuleList[3]
        toggle SR_VisControl.vpiq_axSubControlModuleList[3]
    Button (484,95 117x29), "SubCtrlModule: %s", tooltip "%s", text variable: SR_VisControl.vpq_asSubControlModuleButtonName[4], colour toggle: SR_VisControl.vpq_axSubControlModuleActive[4], invisible if: SR_VisControl.vpq_axSubControlModuleValid[4]=FALSE
        p4168582468: SR_VisControl.vpq_asToolTipSubControlModuleList[4]
        toggle SR_VisControl.vpiq_axSubControlModuleList[4]
    Button (602,95 118x29), "SubCtrlModule: %s", tooltip "%s", text variable: SR_VisControl.vpq_asSubControlModuleButtonName[5], colour toggle: SR_VisControl.vpq_axSubControlModuleActive[5], invisible if: SR_VisControl.vpq_axSubControlModuleValid[5]=FALSE
        p4168582468: SR_VisControl.vpq_asToolTipSubControlModuleList[5]
        toggle SR_VisControl.vpiq_axSubControlModuleList[5]
    Frame (454,127 358x153)
        shows TPL.FR_CurrentModule350x150(i_stCurrentModuleStandardItf := SR_VisControl.vpq_stCurrentModuleStandardInterface)
        p2332068554: SR_VisControl.stCurrentModuleStandardInterface
        p427866952: SR_VisControl.stCurrentModuleStandardInterface
        p2190627833: SR_VisControl.vpq_stCurrentModuleStandardInterface
    Rectangle (30,63 786x216), invisible if: NOT SR_VisControl.vpiq_xShowModuleInterface
    Frame (34,67 380x208), invisible if: NOT SR_VisControl.vpiq_xShowModuleInterface
        shows TPL.FR_StandardModuleInterface380x220(i_stCurrentModuleStandardItf := SR_VisControl.vpq_stCurrentModuleStandardInterface, i_sCurrentModuleReaction := SR_VisControl.vpq_sCurrentModuleReaction, i_udiModuleReactionIndexMin := SR_VisControl.vpq_udiModuleReactionIndexMin, i_axModuleReaction := SR_VisControl.vpq_axModuleReaction, i_udiNumberOfReactions := TPL.Gc_udiMaxNumberOfReactions, iq_xModuleReactionDown := SR_VisControl.vpiq_xModuleReactionDown, iq_xModuleReactionUp := SR_VisControl.vpiq_xModuleReactionUp, iq_diStartStepToSet := SR_VisControl.vpiq_diStartStepToSet, iq_diCmdToSet := SR_VisControl.vpiq_diCmdToSet, iq_xEnableModuleClicked := SR_VisControl.vpiq_xEnableModuleClicked, iq_xSetCmdClicked := SR_VisControl.vpiq_xSetCmdClicked, iq_fbVisContExHandling := SR_VisControl.vpiq_fbVisContExHandling)
        p1094400588: SR_VisControl.IFB_AxisModuleVisController.xCurrentIsOfMyType
        p3339340907: ''
        p1029787830: SR_VisControl.fbVisContExHandling
        p2258115317: SR_VisControl.iModuleErrorReactionIndexMin
        p2777435286: SR_VisControl.axModuleErrorReaction
        p214250784: TPC_Gc_diMaxNumberOfErrorReactions
        p311732222: SR_VisControl.stCurrentModuleStandardInterface
        p640132070: SR_VisControl.xModuleErrorReactionDown
        p4234372197: SR_VisControl.xModuleErrorReactionUp
        p2938682392: SR_VisControl.xEnableModule_Clicked
        p3592490199: SR_VisControl.xSetCmd_Clicked
        p2307280719: SR_VisControl.stCurrentModuleStandardInterface
        p2190627833: SR_VisControl.vpq_stCurrentModuleStandardInterface
    Frame (34,283 778x257), invisible if: SR_VisControl.vpq_stCurrentModuleStandardInterface.q_dwModuleType <> 3
        shows AXM.FR_Details(iq_fbAxisModuleVisController := SR_VisControl.vpiq_fbAxisModuleVisController)
        p334560860: SR_VisControl.IFB_AxisModuleVisController.stCurrentAxisInterface
        p159172089: SR_VisControl.IFB_AxisModuleVisController
        p2012682765: SR_VisControl.stCurrentModuleStandardInterface
        p3545344757: SR_VisControl.stCurrentModuleStandardInterface.i_sModuleName
        p2977392050: SR_VisControl.astEQCMDTable
        p1710090269: SR_VisControl.udiEQTableStepCount
        p3492251336: SR_VisControl.stCurrentModuleStandardInterface.iq_stExt.diActiveStep
        p1862340509: SR_VisControl.sEQCMDTableTitle
        p577637124: SR_VisControl.xDoEnable
        p706691565: NOT SR_VisControl.xEnableCmdTableUp
        p2658775966: NOT SR_VisControl.xEnableCmdTableDown
        p2041874301: SR_VisControl.udiEQTableIndexMin
        p427866952: SR_VisControl.stCurrentModuleStandardInterface
        p4226816124: SR_VisControl.udiEQTableIndexMin
        p2190627833: SR_VisControl.stCurrentModuleStandardInterface
    Frame (34,283 778x257), invisible if: NOT SR_VisControl.vpq_xDisplayCmdTable
        shows TPL.FR_ModuleCommandTable620x250(i_stCurrentModuleStandardItf := SR_VisControl.vpq_stCurrentModuleStandardInterface, i_astActualCmdTable := SR_VisControl.vpq_astActualCmdTableModule, i_udiNumberOfCmdSteps := SR_VisControl.vpq_udiNumberOfCmdStepsModule, i_sCmdTitel := SR_VisControl.vpq_sCmdTitleModule, i_xDoEnable := SR_VisControl.vpq_xDoEnable, i_xDisableScrollUp := SR_VisControl.vpq_xDisableScrollUpModule, i_xDisableScrollDown := SR_VisControl.vpq_xDisableScrollDownModule, iq_udiIndexMin := SR_VisControl.vpiq_udiIndexMinModule)
        p334560860: SR_VisControl.IFB_AxisModuleVisController.stCurrentAxisInterface
        p159172089: SR_VisControl.IFB_AxisModuleVisController
        p2012682765: SR_VisControl.stCurrentModuleStandardInterface
        p3545344757: SR_VisControl.stCurrentModuleStandardInterface.i_sModuleName
        p3492251336: SR_VisControl.vpq_stCurrentModuleStandardInterface.iq_stExt.diActiveStep
        p2041874301: SR_VisControl.udiEQTableIndexMin
        p427866952: SR_VisControl.stCurrentModuleStandardInterface
        p2190627833: SR_VisControl.vpq_stCurrentModuleStandardInterface
    Rectangle (306,720 98x40), "Module Details"
    Frame (819,5 200x430), invisible if: NOT SR_VisControl.vpiq_xShowControlFrame
        shows TPL.FR_MachineControl200x430(i_stMachineItf := SR_VisControl.vpq_stMachineInterface, i_xPrepareActive := G_xPrepareActive, i_xAutoActive := G_xAutoActive, i_xBrakeReleaseActive := G_xBrakeReleaseActive, i_xJogMachineActive := G_xJogMachineActive, i_xManualActive := G_xManualActive, i_xException := SR_VisControl.vpq_xMachineInException, i_dwDiagQuitColor := SR_VisControl.vpq_dwDiagQuitColor, iq_iPositionX := SR_VisControl.vpiq_iPositionX, iq_iPositionY := SR_VisControl.vpiq_iPositionY, iq_xEmergencyEpas := G_xEmergencyEpas, iq_xStartEpas := G_xStartEpas, iq_xStopEpas := G_xStopEpas, iq_xJogForwEpas := G_xJogForwEpas, iq_xJogBackEpas := G_xJogBackEpas, iq_xDoPrepare := G_xDoPrepare, iq_xDoAuto := G_xDoAuto, iq_xDoBrakeRelease := G_xDoBrakeRelease, iq_xDoJogMachine := G_xDoJogMachine, iq_xDoManual := G_xDoManual, iq_xDiagQuitEpas := G_xDiagQuitEpas)
        p1457045297: SR_VisControl.stMachineInterface.stQ.xError
        p1941967854: g_I_xEmergency_Epas
        p2531571229: g_I_xStart_Epas
        p1511842254: g_I_xStop_Epas
        p745511063: g_I_xJogForw_Epas
        p3518271027: g_I_xJogBack_Epas
        p1982879521: g_I_xErrorQuit_Epas
        p3866886353: SR_VisControl.dwErrorQuitColor
        p1761348311: SR_VisControl.vpq_stMachineInterface
        p3560616238: SR_VisControl.vpiq_iPositionX
        p2738717112: SR_VisControl.vpiq_iPositionY
END_VISUALIZATION

// LMC_PacDrive/Application/TemplateFullProgrammingFramework/Visualization/Windows/VIS_ModuleExceptions
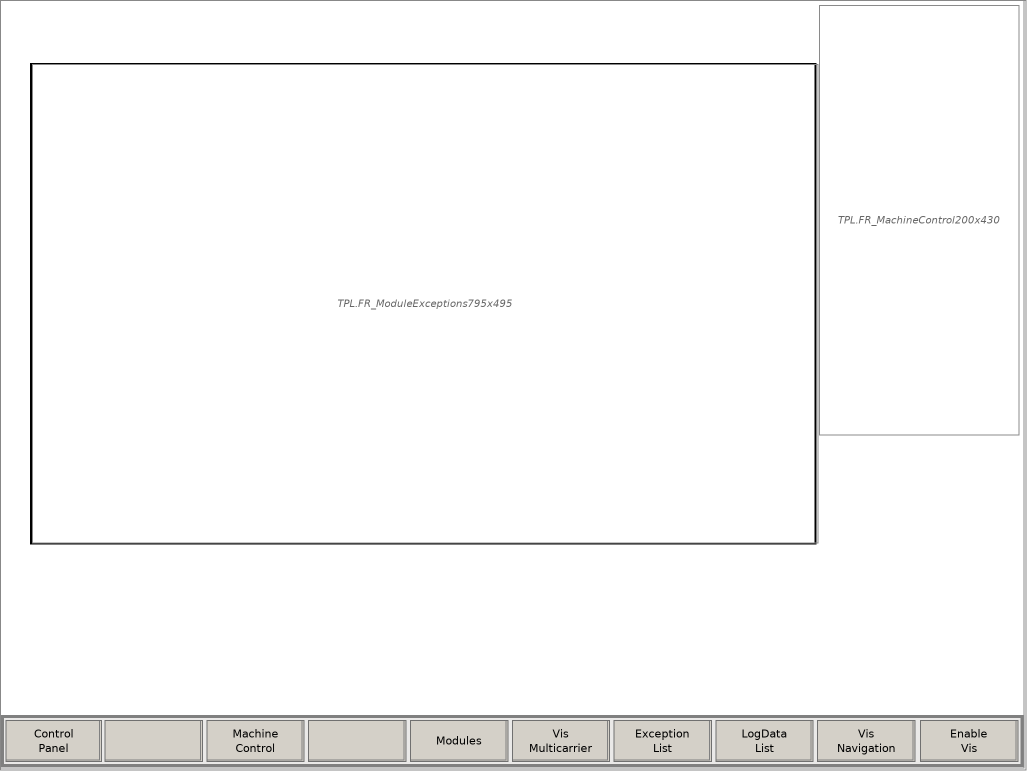
VISUALIZATION VIS_ModuleExceptions  // 1027x771
    Frame (0,0 1024x768)
        shows TPL.FR_Nav1024x768(i_sTitle := 'Template: ModuleExceptions')
    Rectangle (30,63 786x481)
    Frame (32,64 786x479)
        shows TPL.FR_ModuleExceptions795x495(i_stCurrentModuleStandardItf := SR_VisControl.vpq_stCurrentModuleStandardInterface, i_sCurrentModuleReaction := SR_VisControl.vpq_sCurrentModuleReaction, i_udiModuleReactionIndexMin := SR_VisControl.vpq_udiModuleReactionIndexMin, i_axModuleReaction := SR_VisControl.vpq_axModuleReaction, i_udiNumberOfReactions := TPL.Gc_udiMaxNumberOfReactions, iq_xModuleReactionDown := SR_VisControl.vpiq_xModuleReactionDown, iq_xModuleReactionUp := SR_VisControl.vpiq_xModuleReactionUp, iq_diStartStepToSet := SR_VisControl.vpiq_diStartStepToSet, iq_diCmdToSet := SR_VisControl.vpiq_diCmdToSet, iq_xEnableModuleClicked := SR_VisControl.vpiq_xEnableModuleClicked, iq_xSetCmdClicked := SR_VisControl.vpiq_xSetCmdClicked, iq_fbVisContExHandling := SR_VisControl.vpiq_fbVisContExHandling)
        p1094400588: SR_VisControl.IFB_AxisModuleVisController.xCurrentIsOfMyType
        p2258115317: SR_VisControl.iModuleErrorReactionIndexMin
        p2777435286: SR_VisControl.axModuleErrorReaction
        p214250784: TPC_Gc_diMaxNumberOfErrorReactions
        p311732222: SR_VisControl.stCurrentModuleStandardInterface
        p640132070: SR_VisControl.xModuleErrorReactionDown
        p4234372197: SR_VisControl.xModuleErrorReactionUp
        p2938682392: SR_VisControl.xEnableModule_Clicked
        p3592490199: SR_VisControl.xSetCmd_Clicked
        p2307280719: SR_VisControl.stCurrentModuleStandardInterface
        p2190627833: SR_VisControl.vpq_stCurrentModuleStandardInterface
    Frame (1,715 1024x54)
        shows FR_NavigationButtons()
    Frame (819,5 200x430), invisible if: NOT SR_VisControl.vpiq_xShowControlFrame
        shows TPL.FR_MachineControl200x430(i_stMachineItf := SR_VisControl.vpq_stMachineInterface, i_xPrepareActive := G_xPrepareActive, i_xAutoActive := G_xAutoActive, i_xBrakeReleaseActive := G_xBrakeReleaseActive, i_xJogMachineActive := G_xJogMachineActive, i_xManualActive := G_xManualActive, i_xException := SR_VisControl.vpq_xMachineInException, i_dwDiagQuitColor := SR_VisControl.vpq_dwDiagQuitColor, iq_iPositionX := SR_VisControl.vpiq_iPositionX, iq_iPositionY := SR_VisControl.vpiq_iPositionY, iq_xEmergencyEpas := G_xEmergencyEpas, iq_xStartEpas := G_xStartEpas, iq_xStopEpas := G_xStopEpas, iq_xJogForwEpas := G_xJogForwEpas, iq_xJogBackEpas := G_xJogBackEpas, iq_xDoPrepare := G_xDoPrepare, iq_xDoAuto := G_xDoAuto, iq_xDoBrakeRelease := G_xDoBrakeRelease, iq_xDoJogMachine := G_xDoJogMachine, iq_xDoManual := G_xDoManual, iq_xDiagQuitEpas := G_xDiagQuitEpas)
        p1457045297: SR_VisControl.stMachineInterface.stQ.xError
        p1941967854: g_I_xEmergency_Epas
        p2531571229: g_I_xStart_Epas
        p1511842254: g_I_xStop_Epas
        p745511063: g_I_xJogForw_Epas
        p3518271027: g_I_xJogBack_Epas
        p1982879521: g_I_xErrorQuit_Epas
        p3866886353: SR_VisControl.dwErrorQuitColor
        p1761348311: SR_VisControl.vpq_stMachineInterface
        p3560616238: SR_VisControl.vpiq_iPositionX
        p2738717112: SR_VisControl.vpiq_iPositionY
END_VISUALIZATION

